Yaskawa INFORM job: X2_8B-21B(90,180)_HARDOX.JBI

/JOB
//NAME X2_8B-21B(90,180)_HARDOX
///FOLDERNAME X2
//POS
///NPOS 1745,1745,1745,47,0,0
///TOOL 0
///POSTYPE PULSE
///PULSE
C00000=-1415,-134459,-133802,-1969,12985,79332
C00001=-87080,-112473,-103627,-41798,51237,70410
C00002=-91681,-107347,-99471,-39221,49165,68848
C00003=-93439,-105106,-97054,-38371,48113,68361
C00004=-93441,-104864,-95967,-38672,47682,68565
C00005=-93504,-104969,-96260,-38564,47753,68495
C00006=-95585,-102642,-95415,-36914,47385,67494
C00007=-93504,-104969,-96260,-38564,47753,68495
C00008=-87147,-112175,-102116,-42180,50619,70689
C00009=-87145,-119394,-106475,-25944,48524,38750
C00010=-91166,-110510,-101811,-22693,48895,36705
C00011=-92650,-107060,-99920,-21494,49065,35962
C00012=-94767,-104655,-99060,-19829,49198,34943
C00013=-94484,-105085,-99259,-20052,49173,35080
C00014=-93721,-102513,-96995,-20598,49294,35408
C00015=-94484,-105085,-99259,-20052,49173,35080
C00016=-89209,-117497,-105909,-24366,48468,37757
C00017=-93166,-113214,-115710,-1969,57926,79332
C00018=-93710,-106990,-108704,-1652,56802,79139
C00019=-93766,-106412,-107148,-1629,56140,79127
C00020=-93768,-106433,-106329,-1638,55626,79135
C00021=-93918,-105383,-106173,-1535,56065,79069
C00022=-94164,-101296,-104676,-1361,57240,78956
C00023=-93895,-105502,-106499,-1547,56205,79076
C00024=-93151,-113316,-114305,-1998,57010,79354
C00025=-81072,-99391,-111155,-4750,63110,78553
C00026=-81984,-95120,-104767,-4287,61328,78293
C00027=-82103,-94682,-103397,-4241,60705,78273
C00028=-82106,-94924,-102383,-4271,59960,78300
C00029=-82089,-94934,-102578,-4276,60076,78302
C00030=-82803,-90374,-100753,-3806,61258,77993
C00031=-82089,-94934,-102578,-4276,60076,78302
C00032=-81057,-100006,-109908,-4804,62030,78604
C00033=-94004,-119945,-107122,49530,42714,48164
C00034=-93972,-116281,-97047,53343,39935,45878
C00035=-92833,-103149,-88492,51302,40218,47068
C00036=-93174,-100930,-87132,51219,40604,47120
C00037=-93174,-100493,-85792,51770,40220,46795
C00038=-93174,-101015,-87399,51095,40684,47186
C00039=-92955,-97894,-86230,50180,41136,47726
C00040=-93303,-100448,-87190,51023,40860,47230
C00041=-98055,-98607,-86499,53149,43882,46024
C00042=-96642,-96320,-85623,51883,43475,46780
C00043=-95342,-96864,-85830,51299,42647,47109
C00044=-97130,-98187,-86063,52744,43317,46271
C00045=-114545,-105110,-100746,39625,57097,48369
C00046=-113947,-102413,-97570,39574,56382,48359
C00047=-113947,-102278,-96691,39772,56015,48196
C00048=-113346,-99976,-96570,39024,56612,48763
C00049=-112899,-98120,-95866,38597,56823,49078
C00050=-114020,-99555,-96940,39169,57262,48705
C00051=-56302,-84822,-83054,-58022,66572,84014
C00052=-58361,-85953,-83540,-57558,65172,83717
C00053=-56302,-84822,-83054,-58022,66572,84014
C00054=-50122,-85714,-86741,-59061,71306,84454
C00055=-54195,-101901,-111197,-24063,62262,77343
C00056=-67243,-111926,-101536,21450,29925,69540
C00057=-66442,-101704,-94400,19916,30532,70304
C00058=-66308,-99858,-92576,19846,30336,70336
C00059=-66311,-99589,-91307,20230,29731,70137
C00060=-66308,-99960,-93112,19687,30597,70418
C00061=-70591,-100617,-92786,25268,31264,67678
C00062=-70591,-100325,-91437,25755,30647,67424
C00063=-68222,-99738,-91214,22742,30105,68906
C00064=-70591,-100606,-92729,25289,31242,67667
C00065=-66097,-110297,-96199,21577,27345,69446
C00066=-65719,-107666,-92844,21562,26575,69447
C00067=-65848,-106528,-92445,21497,26927,69482
C00068=-65365,-110699,-93884,21743,25627,69354
C00069=-67243,-111926,-101536,21450,29925,69540
C00070=-68963,-41843,-96211,-398,96948,-48811
C00071=-76932,-51697,-92360,2602,89609,-51106
C00072=-71886,-45093,-85416,705,88639,-49643
C00073=-71886,-45937,-84760,705,87803,-49648
C00074=-71886,-44632,-85753,705,89084,-49641
C00075=-68776,-90352,-95136,-4313,51281,-47645
C00076=-68803,-86754,-93636,-4241,52203,-47695
C00077=-68762,-92243,-95906,-4353,50785,-47617
C00078=-77446,-64871,-91176,8832,74282,-49527
C00079=-75907,-64612,-91046,8095,74185,-49034
C00080=-78150,-64967,-91224,9168,74335,-49752
C00081=-78150,-57569,-97635,8943,81990,-49191
C00082=-68963,-41843,-96211,-398,96948,-48811
C00083=-67385,-42511,-92598,-992,94393,-48367
C00084=-66773,-44328,-90253,-1220,92024,-48175
C00085=-66900,-44765,-89647,-1171,91425,-48205
C00086=-66773,-43962,-90441,-1221,92327,-48178
C00087=-69817,-49291,-93527,-72,91467,-49038
C00088=-102407,-61387,-79216,48101,75803,-74984
C00089=-99741,-62884,-79905,47237,74215,-74494
C00090=-102407,-61387,-79216,48101,75803,-74984
C00091=-71396,-101707,-96198,105,39560,-49678
C00092=-71544,-99303,-95354,247,40276,-49753
C00093=-71126,-105930,-97636,-165,38275,-49535
C00094=-74447,-120283,-111838,3099,39699,-51260
C00095=-57750,-84762,-113304,-22338,79933,-80646
C00096=-38298,-117376,-123136,-35520,84192,-83183
C00097=-31003,-114098,-105660,-45955,85390,-81321
C00098=-32496,-116782,-107403,-45795,84408,-81579
C00099=-34116,-118987,-108120,-45640,83088,-81742
C00100=-33779,-118873,-108083,-45678,83285,-81673
C00101=-33779,-118389,-106291,-45736,82677,-81394
C00102=-33116,-116007,-107005,-45711,84199,-81779
C00103=-43122,-77390,-91933,-43525,86904,-87571
C00104=-44353,-78017,-92219,-43231,86215,-87819
C00105=-45440,-79271,-92786,-42975,85486,-87990
C00106=-45102,-79332,-92813,-43057,85636,-87902
C00107=-45102,-79709,-91490,-43095,84888,-87585
C00108=-41853,-68825,-87871,-43817,88900,-87868
C00109=-48095,-31712,-66541,-47290,99218,-86920
C00110=-48762,-33638,-67810,-47108,98755,-86994
C00111=-49503,-35735,-69173,-46902,98237,-87073
C00112=-49389,-35416,-68966,-46933,98317,-87062
C00113=-49389,-36060,-68028,-46814,97684,-86756
C00114=-48487,-32850,-67294,-47182,98948,-86964
C00115=-45126,-25671,-76382,-49967,106798,-89554
C00116=-48508,-32956,-85951,-38791,109748,-85822
C00117=-73491,-115415,-129730,-12591,84406,-82629
C00118=-68604,-111632,-124361,34026,103601,-55041
C00119=-52690,-105642,-114364,31889,95098,-51390
C00120=-51347,-103959,-112740,31690,94497,-51045
C00121=-51347,-104280,-111882,31650,93903,-51212
C00122=-50963,-109237,-114816,31559,93129,-51281
C00123=-54701,-101748,-112541,32228,96580,-51739
C00124=-54580,-102143,-110625,32107,95358,-52042
C00125=-52710,-105778,-111943,31798,93771,-51772
C00126=-54580,-102143,-110625,32107,95358,-52042
C00127=-53574,-106836,-112314,31893,93817,-52092
C00128=-52008,-102475,-110737,31756,94333,-51344
C00129=-53574,-106836,-112314,31893,93817,-52092
C00130=-61074,-96775,-114868,33501,102293,-52496
C00131=-149084,-102156,-129577,22032,95315,-42360
C00132=-128569,-114069,-129208,14930,94899,-36248
C00133=-124702,-111484,-125119,14131,93099,-35189
C00134=-123206,-111006,-122572,13804,91571,-34868
C00135=-123205,-111346,-122108,13798,91123,-34918
C00136=-123169,-110975,-122344,13795,91444,-34870
C00137=-122647,-104244,-120003,13724,93323,-34489
C00138=-123169,-110975,-122344,13795,91444,-34870
C00139=-116503,-109521,-121739,12400,90787,-32743
C00140=-113941,-110266,-121994,11839,90202,-31960
C00141=-116503,-109521,-121739,12400,90787,-32743
C00142=-121595,-114825,-128025,13496,92670,-34216
C00143=-123984,-121300,-124584,22039,85383,-28695
C00144=-118596,-113071,-118409,20758,84424,-26972
C00145=-117828,-112575,-117002,20585,83663,-26833
C00146=-117596,-112721,-116348,20543,83158,-26838
C00147=-117643,-112201,-116474,20543,83493,-26797
C00148=-117846,-106122,-114344,20549,85245,-26570
C00149=-117643,-112201,-116474,20543,83493,-26797
C00150=-125192,-113488,-115877,22341,84450,-29296
C00151=-124919,-116220,-115928,22323,83104,-29449
C00152=-122352,-116155,-116251,21738,82647,-28614
C00153=-124919,-116220,-115928,22323,83104,-29449
C00154=-123984,-121300,-124584,22039,85383,-28695
C00155=-86442,-134681,-133724,-19248,79211,-32552
C00156=-86002,-121949,-124889,-19319,80358,-32581
C00157=-85994,-121959,-123892,-19351,79775,-32484
C00158=-85995,-122137,-123177,-19379,79272,-32404
C00159=-85938,-122450,-123568,-19392,79360,-32398
C00160=-86651,-115539,-121342,-19081,81262,-32951
C00161=-85938,-122450,-123568,-19392,79360,-32398
C00162=-130270,-119263,-121891,15868,79169,-48216
C00163=-132135,-133974,-122544,16883,72658,-49767
C00164=-129371,-136174,-123179,16117,71390,-48932
C00165=-132135,-133974,-122544,16883,72658,-49767
C00166=-120611,-122953,-119681,21560,80854,-22535
C00167=-120610,-122943,-118608,21593,80243,-22645
C00168=-120610,-122853,-116921,21650,79318,-22813
C00169=-120610,-122881,-117271,21638,79506,-22779
C00170=-120610,-122878,-117279,21638,79511,-22778
C00171=-120610,-122881,-117271,21638,79506,-22779
C00172=-120610,-122873,-117198,21640,79468,-22785
C00173=-120610,-122853,-117190,21640,79473,-22785
C00174=-120610,-122873,-117198,21640,79468,-22785
C00175=-120611,-122910,-120952,21522,81605,-22399
C00176=-120612,-120891,-127143,3106,87300,-4415
C00177=-120611,-122177,-124352,3111,84925,-4474
C00178=-120611,-122645,-122467,3116,83527,-4507
C00179=-120611,-122779,-121606,3119,82929,-4523
C00180=-120611,-122697,-122159,3117,83311,-4513
C00181=-120611,-122692,-122166,3117,83318,-4513
C00182=-120611,-122697,-122159,3117,83311,-4513
C00183=-120611,-121412,-126223,3107,86468,-4436
C00184=-96873,-136971,-131305,19961,95014,-27830
C00185=-53188,-122774,-119059,34227,101931,-42117
C00186=-53187,-122644,-116623,34032,100735,-42492
C00187=-53184,-122447,-115007,33919,99986,-42724
C00188=-53180,-122268,-113886,33849,99484,-42877
C00189=-53186,-122531,-115629,33961,100272,-42636
C00190=-53233,-122033,-113114,32057,113501,-44659
C00191=-53229,-122037,-113108,32057,113495,-44659
C00192=-53233,-122033,-113114,32057,113501,-44659
C00193=-53127,-122157,-112856,34567,84618,-41563
C00194=-53132,-122146,-112848,34568,84621,-41564
C00195=-53127,-122157,-112856,34567,84618,-41563
C00196=-53124,-122720,-116247,34514,86111,-41098
C00197=-68676,-133744,-131015,10578,108811,-68614
C00198=-80160,-118182,-130261,-41,125141,-81817
C00199=-80187,-122370,-123619,-70,118933,-81856
C00200=-80183,-122639,-122398,-68,118043,-81854
C00201=-80181,-122756,-121636,-67,117515,-81853
C00202=-80184,-122603,-122588,-68,118179,-81854
C00203=-80182,-122615,-122584,-67,118170,-81853
C00204=-80184,-122603,-122588,-68,118179,-81854
C00205=-80200,-121154,-126606,-75,121396,-81862
C00206=-109164,-117358,-132635,-7350,119146,-48306
C00207=-144183,-119511,-130571,-15498,107286,-7245
C00208=-197934,-122815,-127402,-28006,89082,55776
C00209=-202772,-123889,-124791,-27048,85608,54814
C00210=-204705,-124106,-122314,-26692,83530,54575
C00211=-204705,-124189,-120905,-26732,82711,54762
C00212=-205113,-122699,-120601,-26621,83104,54520
C00213=-208506,-122040,-120392,-25870,82241,53457
C00214=-204510,-125657,-121990,-26775,82699,54838
C00215=-204510,-125393,-124777,-26704,84359,54459
C00216=-217123,-144581,-130617,-26990,80795,43719
C00217=-208514,-157553,-136215,-22784,79668,13108
C00218=-208514,-151468,-127497,-22936,77598,13510
C00219=-209226,-147410,-126429,-22728,78719,13024
C00220=-208514,-151468,-127497,-22936,77598,13510
C00221=-208514,-156517,-134755,-22805,79329,13174
C00222=-187736,-116553,-120968,-36188,98329,31010
C00223=-144869,-104708,-130913,697,92502,-12445
C00224=-97478,-100538,-119508,25976,122096,-72949
C00225=-94415,-115583,-120723,24602,114867,-73486
C00226=-94145,-116737,-119872,24403,113768,-73630
C00227=-94090,-116915,-118863,24267,113100,-73760
C00228=-94227,-118887,-121662,24392,113788,-73658
C00229=-94618,-126072,-123928,23885,111795,-74261
C00230=-93811,-121058,-122280,24303,112998,-73673
C00231=-123165,-134656,-120887,30393,109989,-65140
C00232=-122877,-135920,-118822,30065,108215,-65520
C00233=-120918,-135771,-118381,30417,107339,-64954
C00234=-122877,-135920,-118822,30065,108215,-65520
C00235=-123434,-129548,-123417,31323,113703,-64157
C00236=-126606,-101457,-128935,16844,101795,-36174
C00237=-152779,-135138,-131563,2515,76140,-19155
C00238=-150820,-122490,-124749,1875,78392,-18455
C00239=-150097,-118368,-121531,1645,78513,-18212
C00240=-150095,-118599,-120646,1648,77850,-18220
C00241=-147666,-112236,-119185,871,80184,-17389
C00242=-146670,-110099,-118456,556,80825,-17059
C00243=-148658,-114325,-119887,1186,79554,-17722
C00244=-87079,-91764,-103818,-42328,107533,9448
C00245=-87027,-91004,-101788,-42122,106912,9740
C00246=-89264,-90509,-101588,-42089,105978,9119
C00247=-87027,-91004,-101788,-42122,106912,9740
C00248=-87391,-90282,-107909,-43186,109836,8282
C00249=-92115,-87061,-118989,-19004,94950,-3823
C00250=-78975,-130870,-123203,19746,71053,-12291
C00251=-74317,-97013,-111518,17407,83606,-9286
C00252=-74211,-95430,-110119,17377,83539,-9259
C00253=-74211,-95892,-109317,17397,82840,-9358
C00254=-75305,-113551,-114600,17838,69768,-10493
C00255=-78326,-111051,-111958,19079,70114,-11550
C00256=-78379,-106110,-110225,18937,71523,-11339
C00257=-78263,-116865,-113913,19272,68408,-11810
C00258=-85880,-113569,-112821,22054,71256,-14152
C00259=-85920,-114580,-110580,22309,69503,-14507
C00260=-82054,-114988,-110714,20879,68380,-13249
C00261=-85920,-114580,-110580,22309,69503,-14507
C00262=-78975,-130870,-123203,19746,67177,-12291
C00263=-159950,-115131,-126913,-23322,109234,64770
C00264=-163413,-124246,-126581,-22686,103792,64589
C00265=-164859,-127477,-125491,-22457,101245,64551
C00266=-164857,-127553,-124648,-22406,100728,64651
C00267=-164862,-127370,-126252,-22506,101730,64457
C00268=-158275,-145382,-129341,-21795,96649,67831
C00269=-159759,-153222,-131425,-21726,93697,67826
C00270=-158275,-145382,-129341,-21795,96649,67831
C00271=-157577,-144643,-126617,-21696,95625,68274
C00272=-160219,-140867,-125578,-21868,96138,67212
C00273=-157577,-144643,-126617,-21696,95625,68274
C00274=-152631,-134238,-128202,-21932,102817,68768
C00275=-146941,-123801,-133763,-3444,102850,52685
C00276=-136178,-116173,-124987,31736,84906,22811
C00277=-134413,-106132,-117362,31242,84680,23412
C00278=-134231,-105594,-115694,31219,83968,23286
C00279=-134230,-105863,-115134,31239,83552,23172
C00280=-134007,-104199,-114803,31151,84035,23389
C00281=-133473,-100630,-113499,30965,84737,23780
C00282=-134315,-106237,-115533,31260,83629,23161
C00283=-136272,-117460,-124003,31807,83855,22481
C00284=-136226,-116324,-125056,31750,84893,22789
C00285=-134474,-106353,-117504,31259,84679,23389
C00286=-134275,-105758,-115681,31235,83904,23252
C00287=-134274,-105987,-115198,31252,83547,23154
C00288=-134027,-104733,-115029,31162,83924,23350
C00289=-133465,-100971,-113658,30966,84667,23763
C00290=-134308,-106598,-115693,31262,83551,23142
C00291=-136269,-117902,-124178,31812,83752,22453
C00292=-139753,-124875,-130430,383,75663,-26245
C00293=-143223,-157944,-133481,-5653,58679,-38405
C00294=-140983,-144085,-126452,-6488,61628,-37698
C00295=-140148,-138933,-122655,-6835,62006,-37402
C00296=-140147,-138616,-121921,-6853,61719,-37384
C00297=-140691,-136506,-121897,-6553,62737,-37651
C00298=-138669,-131542,-120459,-7325,64564,-37004
C00299=-140691,-136506,-121897,-6553,62737,-37651
C00300=-145148,-139028,-124584,-4588,62787,-39337
C00301=-159973,-92454,-110285,14523,90938,-48717
C00302=-158765,-97223,-112137,14224,89465,-48492
C00303=-159973,-92454,-110285,14523,90938,-48717
C00304=-164681,-91509,-114703,15696,94847,-49769
C00305=-142525,-105883,-132766,-7713,103357,-60336
C00306=-90751,-115691,-121566,-36045,104861,-61043
C00307=-92920,-122587,-117773,-35137,99152,-60047
C00308=-93124,-123070,-117553,-35091,98753,-60003
C00309=-93124,-123008,-116878,-35050,98435,-59900
C00310=-93160,-123063,-117190,-35068,98555,-59953
C00311=-95752,-125144,-117838,-34977,96947,-60505
C00312=-93160,-123063,-117190,-35068,98555,-59953
C00313=-92038,-109836,-114685,-38536,89453,-57060
C00314=-86810,-100893,-104585,-47463,92019,-56975
C00315=-88449,-102594,-103600,-47188,90148,-56855
C00316=-88449,-102618,-102426,-47172,89639,-56610
C00317=-88449,-102603,-103366,-47184,90046,-56806
C00318=-85133,-99388,-102162,-47637,92393,-56350
C00319=-85168,-99488,-101153,-47595,91912,-56132
C00320=-86978,-101259,-101820,-47360,90627,-56378
C00321=-84037,-98201,-102123,-47804,93363,-56297
C00322=-108771,-112096,-123986,-16313,85813,-59347
C00323=-109769,-112695,-132242,-3132,99947,-61138
C00324=-127404,-127157,-120795,27540,73197,-60883
C00325=-120526,-123085,-115007,25540,69700,-59025
C00326=-119461,-122312,-114032,25210,69192,-58723
C00327=-119461,-122116,-113003,25293,68708,-58832
C00328=-119461,-122312,-114032,25210,69192,-58723
C00329=-94655,-112249,-115827,-1041,75214,-51009
C00330=-93364,-111129,-115444,-1499,75574,-50577
C00331=-121213,-123445,-114215,25873,69302,-59387
C00332=-127714,-127278,-119628,27738,72603,-61150
C00333=-140848,-129628,-128054,17424,84805,-27418
C00334=-127903,-106251,-120637,17388,91568,-15860
C00335=-124887,-98361,-114445,16717,91208,-14907
C00336=-124614,-94849,-112077,16660,91489,-14780
C00337=-117832,-103976,-115449,15062,87719,-13014
C00338=-118209,-109888,-118953,15141,86934,-13233
C00339=-120968,-118649,-124805,15800,86569,-14208
C00340=-112726,-101228,-128594,1890,90279,15897
C00341=-102865,-105549,-130121,-1361,88970,18873
C00342=-85416,-143080,-122146,-23399,58401,32529
C00343=-89847,-131888,-116792,-20882,59491,30436
C00344=-92125,-126361,-114096,-19602,60042,29398
C00345=-92108,-126361,-114086,-19611,60041,29405
C00346=-94963,-119193,-112807,-13876,65309,25883
C00347=-99230,-109273,-111594,-7832,72910,21884
C00348=-97558,-114678,-114533,-8498,72116,22521
C00349=-94805,-124749,-120489,-9597,70928,23580
C00350=-89899,-115674,-129227,-15589,81503,27304
C00351=-94000,-113154,-130859,1035,116659,-75004
C00352=-93721,-118000,-129934,5060,122177,-74127
C00353=-93715,-120352,-127357,4900,119392,-74256
C00354=-95346,-120435,-125547,4467,118331,-74923
C00355=-87734,-123112,-126247,6115,116903,-72103
C00356=-93725,-120284,-127319,4898,119404,-74259
C00357=-93731,-117931,-129895,5059,122189,-74130
C00358=-92605,-107385,-114202,-42080,118626,-78084
C00359=-94957,-117308,-114744,-40643,113912,-77125
C00360=-96859,-119647,-113709,-40343,111617,-77062
C00361=-96820,-119688,-113698,-40330,111613,-77042
C00362=-92369,-120637,-111842,-39132,112371,-75247
C00363=-87506,-133441,-114197,-38673,106213,-75021
C00364=-90618,-118755,-112828,-39302,114392,-75239
C00365=-88476,-109244,-112462,-40625,118981,-76164
C00366=-73726,-95231,-122050,-23824,117115,-78775
C00367=-68964,-113071,-130294,19412,109419,-80322
C00368=-55630,-112625,-122011,35520,97927,-81697
C00369=-52390,-118820,-120628,34805,93310,-81881
C00370=-47869,-106069,-116317,31727,98681,-78960
C00371=-58944,-112669,-113031,37596,97582,-82877
C00372=-56690,-122472,-119439,35129,92879,-83747
C00373=-59872,-116629,-120975,35716,97415,-83571
C00374=-61517,-148095,-119735,48293,75564,-80066
C00375=-55473,-148057,-116974,48060,71191,-79214
C00376=-53771,-146175,-114985,47935,70110,-78894
C00377=-54494,-144748,-112549,48210,69974,-79344
C00378=-55476,-147094,-115701,48129,70996,-79318
C00379=-61520,-147186,-118480,48348,75358,-80173
C00380=-69196,-132761,-125763,48066,87564,-77891
C00381=-67178,-112107,-133350,-9560,121946,-71499
C00382=-53652,-115588,-130730,-10921,119132,-80041
C00383=-53631,-118653,-128170,-10572,116038,-79726
C00384=-49406,-129162,-130962,-9295,109096,-77614
C00385=-56866,-119557,-126808,-10903,114346,-80761
C00386=-54665,-117852,-125979,-10629,114989,-80007
C00387=-57520,-119011,-127190,-3009,114777,-80027
C00388=-59278,-121853,-127991,842,113579,-80159
C00389=-55695,-120300,-124998,1328,112531,-78914
C00390=-53493,-120154,-126714,1639,113579,-78070
C00391=-53512,-117734,-129516,1682,116546,-78033
C00392=-64263,-112177,-127274,18013,116425,-52133
C00393=-53349,-113292,-116223,34708,105130,-41711
C00394=-53347,-113647,-113946,34435,103813,-42137
C00395=-52680,-112871,-112467,34368,103124,-42082
C00396=-58031,-122280,-112065,36284,98076,-45699
C00397=-53343,-113729,-112902,34324,103242,-42318
C00398=-53345,-113489,-115217,34581,104530,-41905
C00399=-83368,-135406,-127982,43757,111124,24122
C00400=-107112,-148704,-121184,48737,110155,73723
C00401=-107085,-142005,-111593,48000,108472,72828
C00402=-107084,-140010,-108705,47787,107957,72557
C00403=-87331,-137626,-115833,38185,104318,80918
C00404=-107143,-152743,-127540,-1092,113262,57657
C00405=-96955,-158208,-128899,-2670,111185,56030
C00406=-107130,-144670,-115956,-40497,90070,47196
C00407=-107133,-145289,-116877,-40503,90261,47122
C00408=-107139,-146938,-119316,-40521,90762,46927
C00409=-81304,-146505,-131302,-46256,99624,33732
C00410=-42290,-135810,-134986,-6789,56953,-43412
C00411=-53482,-111499,-99357,-5283,31563,-44884
C00412=-53488,-110753,-96932,-5448,30458,-44798
C00413=-53106,-110845,-96482,-5998,30161,-44520
C00414=-53143,-110117,-93832,-6189,28906,-44421
C00415=-53188,-109818,-93168,-6175,28651,-44427
C00416=-53095,-108922,-90553,-6542,27518,-44240
C00417=-53472,-108968,-91791,-5862,28222,-44586
C00418=-53466,-109889,-94290,-5675,29282,-44681
C00419=-93748,-113667,-111432,27227,62688,-41579
C00420=-93751,-113561,-109328,27520,61581,-41869
C00421=-94535,-110348,-107800,27711,62471,-41963
C00422=-94560,-109570,-102150,28499,59749,-42715
C00423=-93743,-112935,-104615,28181,59286,-42489
C00424=-93741,-113330,-106821,27872,60309,-42206
C00425=-53707,-103235,-126817,-3349,90409,-72793
C00426=-53694,-107630,-124107,-3352,86490,-72685
C00427=-53689,-108955,-122884,-3357,85060,-72645
C00428=-53697,-108940,-122873,-3354,85062,-72648
C00429=-53721,-108898,-122839,-3346,85062,-72656
C00430=-53729,-108884,-122827,-3345,85059,-72658
C00431=-53735,-107561,-124050,-3339,86489,-72698
C00432=-53748,-103173,-126762,-3336,90406,-72805
C00433=-44251,-68518,-112793,-6305,100072,-70363
C00434=-80270,30794,-42629,-11133,115571,-76543
C00435=-69737,67118,16632,-42575,112328,-80617
C00436=-69636,63823,22197,-49512,110599,-81416
C00437=-67564,55530,12856,-50142,112647,-81508
C00438=-66424,44944,1253,-49852,108764,-84350
C00439=-65618,29495,-14632,-48008,102670,-88237
C00440=-64581,15750,-27557,-48396,103780,-88326
C00441=-64160,11595,-31362,-48525,104124,-88308
C00442=-61878,-10748,-50140,-48981,105285,-87846
C00443=-62672,195,-41330,-51307,112408,-84907
C00444=-58944,10301,-35991,-52571,115494,-84879
C00445=-69716,-6230,-69222,-29298,97742,-75748
C00446=-102330,-22799,-82036,11222,88832,-73278
C00447=-48313,-118911,-129560,19207,92704,-27073
C00448=-53495,-110604,-121584,20154,93282,-28749
C00449=-53898,-112894,-120750,20179,91787,-29140
C00450=-54091,-109968,-119805,20238,92698,-29053
C00451=-54227,-109896,-119946,20266,92849,-29073
C00452=-54259,-112639,-122766,20278,93161,-29031
C00453=-53522,-108468,-123882,20258,95652,-28360
C00454=-66910,-101677,-117691,1645,82254,17515
C00455=-66905,-103395,-115374,1652,79946,17486
C00456=-66559,-103374,-114061,1536,79140,17588
C00457=-66525,-103141,-114029,1523,79241,17602
C00458=-67620,-103650,-114144,1902,79074,17240
C00459=-69811,-106122,-108316,12679,69437,17327
C00460=-66783,-105788,-110032,11324,70201,18483
C00461=-66785,-105108,-112553,11207,72068,18659
C00462=-34610,-119076,-126707,-31995,89279,47352
C00463=-26693,-119602,-105841,-51320,82883,62074
C00464=-26676,-118953,-103885,-51392,82336,62389
C00465=-26611,-118260,-103653,-51381,82509,62328
C00466=-26639,-116853,-99731,-51529,81413,62927
C00467=-26666,-118021,-101324,-51491,81640,62785
C00468=-26683,-118745,-103309,-51412,82173,62476
C00469=-26741,-121947,-116429,-51038,86269,60171
C00470=-80158,-111738,-121779,-46707,81282,-33331
C00471=-80124,-114295,-114082,-47454,77096,-31277
C00472=-80115,-114367,-110881,-47781,75720,-30584
C00473=-79927,-114969,-109893,-47987,75192,-30221
C00474=-79885,-115119,-109957,-48003,75187,-30197
C00475=-80052,-114603,-110983,-47806,75713,-30548
C00476=-80061,-114542,-114188,-47480,77086,-31241
C00477=-80063,-113108,-120040,-30435,104055,-77976
C00478=-80050,-114212,-116860,-30086,101864,-77373
C00479=-80380,-112077,-114717,-30053,101557,-77419
C00480=-79932,-114590,-112006,-35005,85347,-77215
C00481=-79912,-114566,-112044,-35008,85386,-77219
C00482=-80479,-112475,-109427,-36632,80098,-77307
C00483=-80029,-114714,-111597,-36713,80437,-77233
C00484=-82440,-93132,-104306,-35744,84828,-79668
C00485=-83378,-90315,-100640,-35536,83784,-79702
C00486=-86724,-76310,-94495,-34501,85296,-81493
C00487=-81341,-82881,-101909,-35963,88366,-80388
C00488=-80042,-114535,-115070,-36542,82240,-77847
C00489=-80040,-111621,-122742,-8414,85267,-41918
C00490=-80035,-113457,-119567,-8450,82400,-41723
C00491=-81798,-124774,-120168,-7328,73182,-41674
C00492=-80327,-109577,-118133,2572,87034,-53415
C00493=-79380,-112621,-119090,2349,86031,-53125
C00494=-78889,-114029,-118891,6085,83597,-58153
C00495=-80002,-113603,-119620,10752,83390,-63441
C00496=-80006,-103113,-128729,10775,94202,-62513
C00497=-39776,-103787,-110683,-21075,62663,59255
C00498=-39766,-104399,-107995,-21452,60825,59622
C00499=-41663,-99518,-106576,-17765,63773,58656
C00500=-39441,-104963,-106701,-21848,59898,59942
C00501=-39326,-105104,-106740,-21922,59881,59993
C00502=-39744,-104425,-108009,-21464,60826,59630
C00503=-39754,-103814,-110697,-21087,62664,59263
C00504=-47977,-106691,-119962,-23629,83327,62671
C00505=-66867,-99660,-121232,-22132,99220,62132
C00506=-66851,-102572,-118810,-21937,96446,62653
C00507=-74494,-137000,-128982,-14609,78071,53501
C00508=-72467,-138184,-128020,-15181,77278,54315
C00509=-67516,-140688,-126942,-16493,76361,56201
C00510=-43056,-127353,-114280,-36292,85121,62743
C00511=-66851,-103895,-117201,-21852,94891,62938
C00512=-66868,-101493,-119792,-22004,97521,62449
C00513=-74321,-107832,-126985,11736,80239,61811
C00514=-66584,-114412,-108983,34198,49386,64476
C00515=-66581,-113854,-105403,35147,47795,63826
C00516=-59001,-125725,-103773,32485,32454,61113
C00517=-65790,-113886,-101008,36132,45231,63145
C00518=-65568,-123466,-98279,45853,34675,56822
C00519=-65581,-123771,-97752,46366,34344,56544
C00520=-66567,-113311,-102857,35821,46729,63375
C00521=-66569,-114089,-106515,34851,48256,64025
C00522=-66614,-114312,-115902,32344,53032,65825
C00523=-26293,-124733,-123676,35115,86081,77095
C00524=-26278,-124914,-120130,35186,84196,76502
C00525=-26550,-125631,-118910,35285,83385,76132
C00526=-26140,-123752,-118256,35186,83681,76394
C00527=-26301,-124893,-120124,35190,84211,76498
C00528=-26317,-124710,-123669,35119,86096,77090
C00529=-26368,-124828,-121889,39154,95960,78120
C00530=-26350,-124746,-118556,38992,94373,77544
C00531=-26342,-124553,-116950,38932,93670,77290
C00532=-26340,-123995,-113991,38847,92461,76851
C00533=-26347,-124286,-115407,38884,93032,77056
C00534=-26365,-124761,-118865,39006,94524,77592
C00535=-26264,-124528,-116402,47920,86072,68134
C00536=-26249,-123768,-112787,47988,84810,67516
C00537=-26243,-123374,-111311,48022,84325,67278
C00538=-26226,-122772,-109280,48074,83674,66962
C00539=-26232,-123227,-110778,48035,84146,67194
C00540=-26247,-124165,-114452,47952,85370,67795
C00541=-82585,-123093,-118421,52491,64599,59558
C00542=-107155,-118824,-102398,58122,50036,52281
C00543=-107155,-117467,-98958,59145,49269,51564
C00544=-96813,-117817,-104188,42223,47347,50994
C00545=-105933,-121077,-109912,10415,42869,62990
C00546=-105953,-121074,-109843,10442,42831,62975
C00547=-107149,-121400,-109798,11502,42801,62375
C00548=-106717,-121349,-105974,7567,38238,71665
C00549=-107169,-120346,-107141,7797,39493,71540
C00550=-108433,-119625,-117514,7930,46308,71537
C00551=-107111,-122100,-111275,39348,45202,56077
C00552=-107109,-117760,-98763,43179,41028,53713
C00553=-106761,-117495,-97713,43363,40478,53604
C00554=-106458,-119074,-102370,12274,36991,61895
C00555=-94483,-118196,-102129,-13006,37418,75653
C00556=-107097,-114092,-90505,-56996,42891,80282
C00557=-107127,-114270,-91297,-56630,43098,80056
C00558=-101354,-119078,-102486,-55464,49091,79315
C00559=-93612,-109275,-133010,12113,75674,64968
C00560=-74458,-81913,-116300,25886,107898,47202
C00561=-74285,-84923,-113224,25351,104735,46539
C00562=-74085,-86300,-112083,25142,103399,46313
C00563=-71499,-76504,-108067,25490,106819,45523
C00564=-62961,-60085,-100217,24652,107848,48688
C00565=-60437,-59805,-99888,23461,105440,51393
C00566=-60588,-58283,-100875,23679,106756,51616
C00567=-60637,-54628,-103477,24231,109960,52288
C00568=-76657,-70403,-83915,51355,64349,40407
C00569=-74830,-68241,-74355,53953,55282,38932
C00570=-73110,-62379,-68708,53436,54020,39148
C00571=-73126,-62440,-68450,53549,53912,39057
C00572=-36930,-67607,-75173,-26029,44061,77403
C00573=-80523,-89058,-85253,18218,36719,55154
C00574=-82272,-90569,-85112,18702,34759,56728
C00575=-81508,-95500,-88175,18158,33969,56993
C00576=-81043,-103588,-94156,17854,33413,57140
C00577=-82846,-88179,-88219,41798,48730,43563
C00578=-81818,-81213,-82326,41198,48211,43888
C00579=-79663,-80074,-80946,37957,46333,45127
C00580=-64011,-84834,-85332,4259,39755,58703
C00581=-75846,-87347,-86370,15921,40584,52659
C00582=-47572,-67654,-78731,-37306,60592,66422
C00583=-46339,-68382,-80235,-37741,61555,66618
C00584=-42699,-70655,-83815,-39176,63943,67342
C00585=-43803,-67144,-92021,-36183,69839,64523
C00586=-86906,-70734,-117845,25978,101850,24881
C00587=-194376,-118372,-116958,36622,58194,-75254
C00588=-187943,-106127,-101715,33777,52366,-74665
C00589=-187951,-105693,-98645,34509,50978,-75202
C00590=-187954,-105458,-97394,34809,50440,-75417
C00591=-187960,-105469,-97402,34805,50444,-75420
C00592=-187927,-105629,-98482,19599,46235,-60273
C00593=-187923,-105820,-99644,19403,46817,-60144
C00594=-187914,-106157,-102495,18928,48312,-59826
C00595=-188021,-109107,-91072,54887,40419,-77132
C00596=-188025,-108188,-88773,55807,39869,-77674
C00597=-188027,-107805,-87846,56180,39654,-77892
C00598=-188036,-107761,-87717,56242,39627,-77928
C00599=-188035,-108145,-88644,55869,39841,-77710
C00600=-188030,-109068,-90945,54948,40390,-77168
C00601=-188015,-114130,-110744,41340,72657,-75143
C00602=-188018,-113864,-107763,41683,71368,-75679
C00603=-188019,-113684,-106544,41824,70871,-75888
C00604=-188009,-113674,-106577,41816,70886,-75877
C00605=-188008,-113852,-107795,41674,71383,-75668
C00606=-188005,-114114,-110775,41332,72673,-75132
C00607=-187933,-113872,-110928,18210,58720,-57176
C00608=-187882,-113256,-105308,-719,43762,-42538
C00609=-187896,-112711,-102669,-725,42418,-42533
C00610=-187852,-113170,-101841,-775,41671,-42505
C00611=-187778,-112374,-98354,-1639,37547,-42296
C00612=-187899,-111729,-99017,-1491,38283,-42378
C00613=-187886,-112431,-101600,-1465,39511,-42393
C00614=-192869,-127835,-120494,22551,66263,-53872
C00615=-188079,-122619,-114609,40714,83609,-61664
C00616=-188077,-122103,-112045,40794,82601,-62056
C00617=-188097,-121812,-110726,41966,87288,-59780
C00618=-188097,-121769,-110559,41966,87227,-59806
C00619=-188105,-121282,-108770,41980,86589,-60067
C00620=-188106,-121566,-109755,41972,86936,-59927
C00621=-188110,-122188,-112187,41960,87826,-59570
C00622=-188058,-121965,-125191,40549,88870,-59628
C00623=-104402,-90439,-123637,22599,88102,26907
C00624=-80407,-121901,-119741,18448,66455,46046
C00625=-80400,-121844,-116068,18757,64334,45697
C00626=-80358,-121826,-114599,18875,63477,45568
C00627=-79500,-120626,-114191,18436,63629,45929
C00628=-80475,-121542,-115946,18779,64427,45684
C00629=-80482,-121578,-119613,18469,66554,46034
C00630=-85156,-144709,-129107,-21632,59402,64028
C00631=-93856,-120445,-109825,-39450,57641,70752
C00632=-93847,-119691,-106928,-40019,56559,71233
C00633=-86628,-99816,-98593,-45940,69277,74290
C00634=-86043,-99167,-98859,-45014,69635,74495
C00635=-83318,-93529,-94650,-47165,68336,75996
C00636=-93680,-116508,-100417,-40719,46210,72415
C00637=-93820,-118277,-102341,-40471,46353,72255
C00638=-93828,-119232,-105178,-39715,47322,71755
C00639=-93822,-120125,-107980,-28359,52237,38282
C00640=-93816,-119582,-106091,-28689,51458,38525
C00641=-93813,-119346,-105328,-28822,51152,38622
C00642=-93805,-118409,-102529,-29499,49391,39302
C00643=-93820,-119862,-107056,-29266,59584,40856
C00644=-93823,-120114,-107958,-29147,59957,40747
C00645=-93830,-120670,-110185,-28854,60909,40473
C00646=-63807,-119595,-131717,-32346,77391,31957
C00647=-66677,-122882,-119460,-9954,65715,-31882
C00648=-66675,-122709,-116301,-10101,63887,-31721
C00649=-66675,-122586,-115330,-10147,63360,-31673
C00650=-66678,-122782,-121307,9429,81851,-37654
C00651=-66765,-122962,-121469,9451,81867,-37681
C00652=-66675,-122328,-113778,33290,107246,-42961
C00653=-66675,-122499,-114776,33395,107690,-42822
C00654=-66677,-122795,-117228,33681,108831,-42458
C00655=-66720,-122114,-124411,34847,112827,-41144
C00656=-15972,-110889,-128286,-10965,59905,-43045
C00657=-1415,-134459,-133802,-1969,12985,79332
C00658=-87080,-112473,-103627,-41798,51237,70410
C00659=-91681,-107347,-99471,-39221,49165,68848
C00660=-93439,-105106,-97054,-38371,48113,68361
C00661=-93441,-104864,-95967,-38672,47682,68565
C00662=-93504,-104969,-96260,-38564,47753,68495
C00663=-95585,-102642,-95415,-36914,47385,67494
C00664=-93504,-104969,-96260,-38564,47753,68495
C00665=-87147,-112175,-102116,-42180,50619,70689
C00666=-87145,-119394,-106475,-25944,48524,38750
C00667=-91166,-110510,-101811,-22693,48895,36705
C00668=-92650,-107060,-99920,-21494,49065,35962
C00669=-94767,-104655,-99060,-19829,49198,34943
C00670=-94484,-105085,-99259,-20052,49173,35080
C00671=-93721,-102513,-96995,-20598,49294,35408
C00672=-94484,-105085,-99259,-20052,49173,35080
C00673=-89209,-117497,-105909,-24366,48468,37757
C00674=-93166,-113214,-115710,-1969,57926,79332
C00675=-122366,-117496,-112293,16338,56235,67679
C00676=-123456,-103417,-106445,16337,59944,67813
C00677=-123456,-103539,-105172,16474,59132,67689
C00678=-123456,-103531,-105272,16463,59195,67698
C00679=-123128,-98284,-103303,16044,60561,68033
C00680=-123156,-99911,-105489,15984,61057,68095
C00681=-93710,-106990,-108704,-1652,56802,79139
C00682=-93766,-106412,-107148,-1629,56140,79127
C00683=-93768,-106433,-106329,-1638,55626,79135
C00684=-93918,-105383,-106173,-1535,56065,79069
C00685=-94164,-101296,-104676,-1361,57240,78956
C00686=-93895,-105502,-106499,-1547,56205,79076
C00687=-93151,-113316,-114305,-1998,57010,79354
C00688=-81072,-99391,-111155,-4750,63110,78553
C00689=-81984,-95120,-104767,-4287,61328,78293
C00690=-82103,-94682,-103397,-4241,60705,78273
C00691=-82106,-94924,-102383,-4271,59960,78300
C00692=-82089,-94934,-102578,-4276,60076,78302
C00693=-82803,-90374,-100753,-3806,61258,77993
C00694=-82089,-94934,-102578,-4276,60076,78302
C00695=-81057,-100006,-109908,-4804,62030,78604
C00696=-94004,-119945,-107122,49530,42714,48164
C00697=-93972,-116281,-97047,53343,39935,45878
C00698=-92833,-103149,-88492,51302,40218,47068
C00699=-93174,-100930,-87132,51219,40604,47120
C00700=-93174,-100493,-85792,51770,40220,46795
C00701=-93174,-101015,-87399,51095,40684,47186
C00702=-92955,-97894,-86230,50180,41136,47726
C00703=-93303,-100448,-87190,51023,40860,47230
C00704=-98055,-98607,-86499,53149,43882,46024
C00705=-96642,-96320,-85623,51883,43475,46780
C00706=-95342,-96864,-85830,51299,42647,47109
C00707=-97130,-98187,-86063,52744,43317,46271
C00708=-114545,-105110,-100746,39625,57097,48369
C00709=-113947,-102413,-97570,39574,56382,48359
C00710=-113947,-102278,-96691,39772,56015,48196
C00711=-113346,-99976,-96570,39024,56612,48763
C00712=-112899,-98120,-95866,38597,56823,49078
C00713=-114020,-99555,-96940,39169,57262,48705
C00714=-56302,-84822,-83054,-58022,66572,84014
C00715=-58361,-85953,-83540,-57558,65172,83717
C00716=-56302,-84822,-83054,-58022,66572,84014
C00717=-50122,-85714,-86741,-59061,71306,84454
C00718=-54195,-101901,-111197,-24063,62262,77343
C00719=-67243,-111926,-101536,21450,29925,69540
C00720=-66442,-101704,-94400,19916,30532,70304
C00721=-66308,-99858,-92576,19846,30336,70336
C00722=-66311,-99589,-91307,20230,29731,70137
C00723=-66308,-99960,-93112,19687,30597,70418
C00724=-70591,-100617,-92786,25268,31264,67678
C00725=-70591,-100325,-91437,25755,30647,67424
C00726=-68222,-99738,-91214,22742,30105,68906
C00727=-70591,-100606,-92729,25289,31242,67667
C00728=-66097,-110297,-96199,21577,27345,69446
C00729=-65719,-107666,-92844,21562,26575,69447
C00730=-65848,-106528,-92445,21497,26927,69482
C00731=-65365,-110699,-93884,21743,25627,69354
C00732=-67243,-111926,-101536,21450,29925,69540
C00733=-68963,-41843,-96211,-398,96948,-48811
C00734=-76932,-51697,-92360,2602,89609,-51106
C00735=-71886,-45093,-85416,705,88639,-49643
C00736=-71886,-45937,-84760,705,87803,-49648
C00737=-71886,-44632,-85753,705,89084,-49641
C00738=-68776,-90352,-95136,-4313,51281,-47645
C00739=-68803,-86754,-93636,-4241,52203,-47695
C00740=-68762,-92243,-95906,-4353,50785,-47617
C00741=-77446,-64871,-91176,8832,74282,-49527
C00742=-75907,-64612,-91046,8095,74185,-49034
C00743=-78150,-64967,-91224,9168,74335,-49752
C00744=-78150,-57569,-97635,8943,81990,-49191
C00745=-68963,-41843,-96211,-398,96948,-48811
C00746=-67385,-42511,-92598,-992,94393,-48367
C00747=-66773,-44328,-90253,-1220,92024,-48175
C00748=-66900,-44765,-89647,-1171,91425,-48205
C00749=-66773,-43962,-90441,-1221,92327,-48178
C00750=-69817,-49291,-93527,-72,91467,-49038
C00751=-102407,-61387,-79216,48101,75803,-74984
C00752=-99741,-62884,-79905,47237,74215,-74494
C00753=-102407,-61387,-79216,48101,75803,-74984
C00754=-71396,-101707,-96198,105,39560,-49678
C00755=-71544,-99303,-95354,247,40276,-49753
C00756=-71126,-105930,-97636,-165,38275,-49535
C00757=-74447,-120283,-111838,3099,39699,-51260
C00758=-57750,-84762,-113304,-22338,79933,-80646
C00759=-38298,-117376,-123136,-35520,84192,-83183
C00760=-31003,-114098,-105660,-45955,85390,-81321
C00761=-32496,-116782,-107403,-45795,84408,-81579
C00762=-34116,-118987,-108120,-45640,83088,-81742
C00763=-33779,-118873,-108083,-45678,83285,-81673
C00764=-33779,-118389,-106291,-45736,82677,-81394
C00765=-33116,-116007,-107005,-45711,84199,-81779
C00766=-43122,-77390,-91933,-43525,86904,-87571
C00767=-44353,-78017,-92219,-43231,86215,-87819
C00768=-45440,-79271,-92786,-42975,85486,-87990
C00769=-45102,-79332,-92813,-43057,85636,-87902
C00770=-45102,-79709,-91490,-43095,84888,-87585
C00771=-41853,-68825,-87871,-43817,88900,-87868
C00772=-48095,-31712,-66541,-47290,99218,-86920
C00773=-48762,-33638,-67810,-47108,98755,-86994
C00774=-49503,-35735,-69173,-46902,98237,-87073
C00775=-49389,-35416,-68966,-46933,98317,-87062
C00776=-49389,-36060,-68028,-46814,97684,-86756
C00777=-48487,-32850,-67294,-47182,98948,-86964
C00778=-45126,-25671,-76382,-49967,106798,-89554
C00779=-48508,-32956,-85951,-38791,109748,-85822
C00780=-73491,-115415,-129730,-12591,84406,-82629
C00781=-68604,-111632,-124361,34026,103601,-55041
C00782=-52690,-105642,-114364,31889,95098,-51390
C00783=-50963,-109289,-114635,31553,93010,-51314
C00784=-50968,-109442,-114037,31534,92627,-51422
C00785=-50963,-109237,-114816,31559,93129,-51281
C00786=-54701,-101748,-112541,32228,96580,-51739
C00787=-54580,-102143,-110625,32107,95358,-52042
C00788=-52710,-105778,-111943,31798,93771,-51772
C00789=-54580,-102143,-110625,32107,95358,-52042
C00790=-53574,-106836,-112314,31893,93817,-52092
C00791=-52008,-102475,-110737,31756,94333,-51344
C00792=-53574,-106836,-112314,31893,93817,-52092
C00793=-61074,-96775,-114868,33501,102293,-52496
C00794=-149084,-102156,-129577,22032,95315,-42360
C00795=-128569,-114069,-129208,14930,94899,-36248
C00796=-124702,-111484,-125119,14131,93099,-35189
C00797=-123206,-111006,-122572,13804,91571,-34868
C00798=-123205,-111346,-122108,13798,91123,-34918
C00799=-123169,-110975,-122344,13795,91444,-34870
C00800=-122647,-104244,-120003,13724,93323,-34489
C00801=-123169,-110975,-122344,13795,91444,-34870
C00802=-116503,-109521,-121739,12400,90787,-32743
C00803=-113941,-110266,-121994,11839,90202,-31960
C00804=-116503,-109521,-121739,12400,90787,-32743
C00805=-121595,-114825,-128025,13496,92670,-34216
C00806=-123984,-121300,-124584,22039,85383,-28695
C00807=-118596,-113071,-118409,20758,84424,-26972
C00808=-117828,-112575,-117002,20585,83663,-26833
C00809=-117596,-112721,-116348,20543,83158,-26838
C00810=-117643,-112201,-116474,20543,83493,-26797
C00811=-117846,-106122,-114344,20549,85245,-26570
C00812=-117643,-112201,-116474,20543,83493,-26797
C00813=-125192,-113488,-115877,22341,84450,-29296
C00814=-124919,-116220,-115928,22323,83104,-29449
C00815=-122352,-116155,-116251,21738,82647,-28614
C00816=-124919,-116220,-115928,22323,83104,-29449
C00817=-123984,-121300,-124584,22039,85383,-28695
C00818=-86442,-134681,-133724,-19248,79211,-32552
C00819=-86002,-121949,-124889,-19319,80358,-32581
C00820=-85994,-121959,-123892,-19351,79775,-32484
C00821=-85995,-122137,-123177,-19379,79272,-32404
C00822=-85938,-122450,-123568,-19392,79360,-32398
C00823=-86651,-115539,-121342,-19081,81262,-32951
C00824=-85938,-122450,-123568,-19392,79360,-32398
C00825=-130270,-119263,-121891,15868,79169,-48216
C00826=-132135,-133974,-122544,16883,72658,-49767
C00827=-129371,-136174,-123179,16117,71390,-48932
C00828=-132135,-133974,-122544,16883,72658,-49767
C00829=-120611,-122953,-119681,21560,80854,-22535
C00830=-120610,-122943,-118608,21593,80243,-22645
C00831=-120610,-122853,-116921,21650,79318,-22813
C00832=-120610,-122881,-117271,21638,79506,-22779
C00833=-120610,-122878,-117279,21638,79511,-22778
C00834=-120610,-122881,-117271,21638,79506,-22779
C00835=-120610,-122873,-117198,21640,79468,-22785
C00836=-120610,-122853,-117190,21640,79473,-22785
C00837=-120610,-122873,-117198,21640,79468,-22785
C00838=-120611,-122910,-120952,21522,81605,-22399
C00839=-86002,-120340,-127953,-19212,82925,-32989
C00840=-85994,-121959,-123892,-19351,79775,-32484
C00841=-85995,-122137,-123177,-19379,79272,-32404
C00842=-85938,-122450,-123568,-19392,79360,-32398
C00843=-86651,-115539,-121342,-19081,81262,-32951
C00844=-85938,-122450,-123568,-19392,79360,-32398
C00845=-130270,-119263,-121891,15868,79169,-48216
C00846=-132135,-133974,-122544,16883,72658,-49767
C00847=-129371,-136174,-123179,16117,71390,-48932
C00848=-132135,-133974,-122544,16883,72658,-49767
C00849=-120612,-120891,-127143,3106,87300,-4415
C00850=-120611,-122177,-124352,3111,84925,-4474
C00851=-120611,-122645,-122467,3116,83527,-4507
C00852=-120611,-122779,-121606,3119,82929,-4523
C00853=-120611,-122697,-122159,3117,83311,-4513
C00854=-120611,-122692,-122166,3117,83318,-4513
C00855=-120611,-122697,-122159,3117,83311,-4513
C00856=-120611,-121412,-126223,3107,86468,-4436
C00857=-120611,-118807,-129728,3107,89959,-4350
C00858=-120605,-132560,-136700,3104,87187,-4416
C00859=-53188,-122658,-121398,34453,103181,-41719
C00860=-53187,-122644,-116623,34032,100735,-42492
C00861=-53184,-122447,-115007,33919,99986,-42724
C00862=-53180,-122268,-113886,33849,99484,-42877
C00863=-53186,-122531,-115629,33961,100272,-42636
C00864=-53233,-122033,-113114,32057,113501,-44659
C00865=-53229,-122037,-113108,32057,113495,-44659
C00866=-53233,-122033,-113114,32057,113501,-44659
C00867=-53127,-122157,-112856,34567,84618,-41563
C00868=-53132,-122146,-112848,34568,84621,-41564
C00869=-53127,-122157,-112856,34567,84618,-41563
C00870=-53124,-122720,-116247,34514,86111,-41098
C00871=-61684,-126457,-131749,21672,103686,-55019
C00872=-68676,-133744,-131015,10578,108811,-68614
C00873=-80160,-118182,-130261,-41,125141,-81817
C00874=-80187,-122370,-123619,-70,118933,-81856
C00875=-80183,-122639,-122398,-68,118043,-81854
C00876=-80181,-122756,-121636,-67,117515,-81853
C00877=-80184,-122603,-122588,-68,118179,-81854
C00878=-80182,-122615,-122584,-67,118170,-81853
C00879=-80184,-122603,-122588,-68,118179,-81854
C00880=-80200,-121154,-126606,-75,121396,-81862
C00881=-109164,-117358,-132635,-7350,119146,-48306
C00882=-144183,-119511,-130571,-15498,107286,-7245
C00883=-197934,-122815,-127402,-28006,89082,55776
C00884=-202772,-123889,-124791,-27048,85608,54814
C00885=-204705,-124106,-122314,-26692,83530,54575
C00886=-204705,-124189,-120905,-26732,82711,54762
C00887=-205113,-122699,-120601,-26621,83104,54520
C00888=-208506,-122040,-120392,-25870,82241,53457
C00889=-204510,-125657,-121990,-26775,82699,54838
C00890=-204510,-125393,-124777,-26704,84359,54459
C00891=-217123,-144581,-130617,-26990,80795,43719
C00892=-208514,-157553,-136215,-22784,79668,13108
C00893=-208134,-153606,-128050,-23049,77001,13769
C00894=-209226,-147410,-126429,-22728,78719,13024
C00895=-208514,-151468,-127497,-22936,77598,13510
C00896=-208514,-156517,-134755,-22805,79329,13174
C00897=-197934,-122815,-127402,-28006,89082,55776
C00898=-202772,-123889,-124791,-27048,85608,54814
C00899=-204705,-124106,-122314,-26692,83530,54575
C00900=-204705,-124189,-120905,-26732,82711,54762
C00901=-205113,-122699,-120601,-26621,83104,54520
C00902=-208506,-122040,-120392,-25870,82241,53457
C00903=-204510,-125657,-121990,-26775,82699,54838
C00904=-204510,-125393,-124777,-26704,84359,54459
C00905=-217123,-144581,-130617,-26990,80795,43719
C00906=-216657,-144339,-132121,-20327,83655,24427
C00907=-208514,-151468,-127497,-22936,77598,13510
C00908=-209226,-147410,-126429,-22728,78719,13024
C00909=-208514,-151468,-127497,-22936,77598,13510
C00910=-208514,-156517,-134755,-22805,79329,13174
C00911=-187736,-116553,-120968,-36188,98329,31010
C00912=-144869,-104708,-130913,697,92502,-12445
C00913=-97478,-100538,-119508,25976,122096,-72949
C00914=-94415,-115583,-120723,24602,114867,-73486
C00915=-94145,-116737,-119872,24403,113768,-73630
C00916=-94090,-116915,-118863,24267,113100,-73760
C00917=-94227,-118887,-121662,24392,113788,-73658
C00918=-94618,-126072,-123928,23885,111795,-74261
C00919=-93811,-121058,-122280,24303,112998,-73673
C00920=-123165,-134656,-120887,30393,109989,-65140
C00921=-122877,-135920,-118822,30065,108215,-65520
C00922=-120918,-135771,-118381,30417,107339,-64954
C00923=-122877,-135920,-118822,30065,108215,-65520
C00924=-123434,-129548,-123417,31323,113703,-64157
C00925=-126606,-101457,-128935,16844,101795,-36174
C00926=-152779,-135138,-131563,2515,76140,-19155
C00927=-150820,-122490,-124749,1875,78392,-18455
C00928=-150097,-118368,-121531,1645,78513,-18212
C00929=-150095,-118599,-120646,1648,77850,-18220
C00930=-147666,-112236,-119185,871,80184,-17389
C00931=-146670,-110099,-118456,556,80825,-17059
C00932=-148658,-114325,-119887,1186,79554,-17722
C00933=-87079,-91764,-103818,-42328,107533,9448
C00934=-87027,-91004,-101788,-42122,106912,9740
C00935=-89264,-90509,-101588,-42089,105978,9119
C00936=-87027,-91004,-101788,-42122,106912,9740
C00937=-87391,-90282,-107909,-43186,109836,8282
C00938=-92115,-87061,-118989,-19004,94950,-3823
C00939=-78975,-130870,-123203,19746,71053,-12291
C00940=-74317,-97013,-111518,17407,83606,-9286
C00941=-74211,-95430,-110119,17377,83539,-9259
C00942=-74211,-95892,-109317,17397,82840,-9358
C00943=-75305,-113551,-114600,17838,69768,-10493
C00944=-78326,-111051,-111958,19079,70114,-11550
C00945=-78379,-106110,-110225,18937,71523,-11339
C00946=-78263,-116865,-113913,19272,68408,-11810
C00947=-85880,-113569,-112821,22054,71256,-14152
C00948=-85920,-114580,-110580,22309,69503,-14507
C00949=-82054,-114988,-110714,20879,68380,-13249
C00950=-85920,-114580,-110580,22309,69503,-14507
C00951=-78975,-130870,-123203,19746,67177,-12291
C00952=-159950,-115131,-126913,-23322,109234,64770
C00953=-163413,-124246,-126581,-22686,103792,64589
C00954=-164859,-127477,-125491,-22457,101245,64551
C00955=-164857,-127553,-124648,-22406,100728,64651
C00956=-164862,-127370,-126252,-22506,101730,64457
C00957=-158275,-145382,-129341,-21795,96649,67831
C00958=-159759,-153222,-131425,-21726,93697,67826
C00959=-158275,-145382,-129341,-21795,96649,67831
C00960=-157577,-144643,-126617,-21696,95625,68274
C00961=-160219,-140867,-125578,-21868,96138,67212
C00962=-157577,-144643,-126617,-21696,95625,68274
C00963=-152631,-134238,-128202,-21932,102817,68768
C00964=-146941,-123801,-133763,-3444,102850,52685
C00965=-136178,-116173,-124987,31736,84906,22811
C00966=-134413,-106132,-117362,31242,84680,23412
C00967=-134231,-105594,-115694,31219,83968,23286
C00968=-134230,-105863,-115134,31239,83552,23172
C00969=-134007,-104199,-114803,31151,84035,23389
C00970=-133473,-100630,-113499,30965,84737,23780
C00971=-134315,-106237,-115533,31260,83629,23161
C00972=-136272,-117460,-124003,31807,83855,22481
C00973=-136226,-116324,-125056,31750,84893,22789
C00974=-134474,-106353,-117504,31259,84679,23389
C00975=-134275,-105758,-115681,31235,83904,23252
C00976=-134274,-105987,-115198,31252,83547,23154
C00977=-134027,-104733,-115029,31162,83924,23350
C00978=-133465,-100971,-113658,30966,84667,23763
C00979=-134308,-106598,-115693,31262,83551,23142
C00980=-178993,-121773,-123174,38769,99022,10273
C00981=-175539,-115427,-119854,38657,98481,11541
C00982=-175539,-115857,-118311,38525,97555,11203
C00983=-175539,-115829,-118427,38535,97623,11227
C00984=-173168,-111114,-116839,38478,97741,12267
C00985=-174072,-113112,-119760,38657,98741,12252
C00986=-136269,-117902,-124178,31812,83752,22453
C00987=-139753,-124875,-130430,383,75663,-26245
C00988=-143223,-157944,-133481,-5653,58679,-38405
C00989=-140983,-144085,-126452,-6488,61628,-37698
C00990=-140148,-138933,-122655,-6835,62006,-37402
C00991=-140147,-138616,-121921,-6853,61719,-37384
C00992=-140691,-136506,-121897,-6553,62737,-37651
C00993=-138669,-131542,-120459,-7325,64564,-37004
C00994=-140691,-136506,-121897,-6553,62737,-37651
C00995=-145148,-139028,-124584,-4588,62787,-39337
C00996=-159973,-92454,-110285,14523,90938,-48717
C00997=-158765,-97223,-112137,14224,89465,-48492
C00998=-159973,-92454,-110285,14523,90938,-48717
C00999=-164681,-91509,-114703,15696,94847,-49769
C01000=-142525,-105883,-132766,-7713,103357,-60336
C01001=-90751,-115691,-121566,-36045,104861,-61043
C01002=-92920,-122587,-117773,-35137,99152,-60047
C01003=-93124,-123070,-117553,-35091,98753,-60003
C01004=-93124,-123008,-116878,-35050,98435,-59900
C01005=-93160,-123063,-117190,-35068,98555,-59953
C01006=-95752,-125144,-117838,-34977,96947,-60505
C01007=-93160,-123063,-117190,-35068,98555,-59953
C01008=-92038,-109836,-114685,-38536,89453,-57060
C01009=-86810,-100893,-104585,-47463,92019,-56975
C01010=-88449,-102594,-103600,-47188,90148,-56855
C01011=-88449,-102618,-102426,-47172,89639,-56610
C01012=-88449,-102603,-103366,-47184,90046,-56806
C01013=-85133,-99388,-102162,-47637,92393,-56350
C01014=-85168,-99488,-101153,-47595,91912,-56132
C01015=-86978,-101259,-101820,-47360,90627,-56378
C01016=-84037,-98201,-102123,-47804,93363,-56297
C01017=-108771,-112096,-123986,-16313,85813,-59347
C01018=-109769,-112695,-132242,-3132,99947,-61138
C01019=-127404,-127157,-120795,27540,73197,-60883
C01020=-120526,-123085,-115007,25540,69700,-59025
C01021=-119461,-122312,-114032,25210,69192,-58723
C01022=-119461,-122116,-113003,25293,68708,-58832
C01023=-119461,-122312,-114032,25210,69192,-58723
C01024=-94655,-112249,-115827,-1041,75214,-51009
C01025=-93364,-111129,-115444,-1499,75574,-50577
C01026=-121213,-123445,-114215,25873,69302,-59387
C01027=-127714,-127278,-119628,27738,72603,-61150
C01028=-140848,-129628,-128054,17424,84805,-27418
C01029=-127903,-106251,-120637,17388,91568,-15860
C01030=-124887,-98361,-114445,16717,91208,-14907
C01031=-124532,-94860,-112080,16625,91471,-14753
C01032=-117832,-103976,-115449,15062,87719,-13014
C01033=-118209,-109888,-118953,15141,86934,-13233
C01034=-120968,-118649,-124805,15800,86569,-14208
C01035=-112726,-101228,-128594,1890,90279,15897
C01036=-102865,-105549,-130121,-1361,88970,18873
C01037=-85416,-143080,-122146,-23399,58401,32529
C01038=-89847,-131888,-116792,-20882,59491,30436
C01039=-92125,-126361,-114096,-19602,60042,29398
C01040=-92108,-126361,-114086,-19611,60041,29405
C01041=-94963,-119193,-112807,-13876,65309,25883
C01042=-99230,-109273,-111594,-7832,72910,21884
C01043=-97558,-114678,-114533,-8498,72116,22521
C01044=-94805,-124749,-120489,-9597,70928,23580
C01045=-89899,-115674,-129227,-15589,81503,27304
C01046=-94000,-113154,-130859,1035,116659,-75004
C01047=-93721,-118000,-129934,5060,122177,-74127
C01048=-93715,-120352,-127357,4900,119392,-74256
C01049=-95346,-120435,-125547,4467,118331,-74923
C01050=-87734,-123112,-126247,6115,116903,-72103
C01051=-93725,-120284,-127319,4898,119404,-74259
C01052=-93731,-117931,-129895,5059,122189,-74130
C01053=-92605,-107385,-114202,-42080,118626,-78084
C01054=-94957,-117308,-114744,-40643,113912,-77125
C01055=-96859,-119647,-113709,-40343,111617,-77062
C01056=-96820,-119688,-113698,-40330,111613,-77042
C01057=-92369,-120637,-111842,-39132,112371,-75247
C01058=-87506,-133441,-114197,-38673,106213,-75021
C01059=-90618,-118755,-112828,-39302,114392,-75239
C01060=-88476,-109244,-112462,-40625,118981,-76164
C01061=-73726,-95231,-122050,-23824,117115,-78775
C01062=-68964,-113071,-130294,19412,109419,-80322
C01063=-55630,-112625,-122011,35520,97927,-81697
C01064=-52390,-118820,-120628,34805,93310,-81881
C01065=-53603,-103093,-112884,36459,100480,-79984
C01066=-59619,-117562,-114740,37336,94951,-84077
C01067=-56690,-122472,-119439,35129,92879,-83747
C01068=-59872,-116629,-120975,35716,97415,-83571
C01069=-61517,-148095,-119735,48293,75564,-80066
C01070=-55473,-148057,-116974,48060,71191,-79214
C01071=-53771,-146175,-114985,47935,70110,-78894
C01072=-54494,-144748,-112549,48210,69974,-79344
C01073=-55476,-147094,-115701,48129,70996,-79318
C01074=-61520,-147186,-118480,48348,75358,-80173
C01075=-87978,-108563,-128727,6750,125872,-71649
C01076=-93715,-120352,-127357,4900,119392,-74256
C01077=-94748,-123674,-126724,4558,117361,-74733
C01078=-87347,-125535,-127084,6155,116151,-72000
C01079=-93725,-120284,-127319,4898,119404,-74259
C01080=-93731,-117931,-129895,5059,122189,-74130
C01081=-92605,-107385,-114202,-42080,118626,-78084
C01082=-94957,-117308,-114744,-40643,113912,-77125
C01083=-96514,-122009,-114462,-40074,111194,-76723
C01084=-96015,-122145,-114253,-39942,111269,-76518
C01085=-92174,-122830,-112540,-38890,111906,-74970
C01086=-86945,-136787,-114983,-38317,105485,-74493
C01087=-90618,-118755,-112828,-39302,114392,-75239
C01088=-88476,-109244,-112462,-40625,118981,-76164
C01089=-73726,-95231,-122050,-23824,117115,-78775
C01090=-68964,-113071,-130294,19412,109419,-80322
C01091=-55630,-112625,-122011,35520,97927,-81697
C01092=-52390,-118820,-120628,34805,93310,-81881
C01093=-47304,-107066,-116669,31636,98225,-78870
C01094=-58547,-113359,-113266,37552,97245,-82829
C01095=-56690,-122472,-119439,35129,92879,-83747
C01096=-59872,-116629,-120975,35716,97415,-83571
C01097=-61517,-148095,-119735,48293,75564,-80066
C01098=-55473,-148057,-116974,48060,71191,-79214
C01099=-53043,-147267,-115261,47953,69457,-78858
C01100=-53748,-146178,-113424,48182,69442,-79233
C01101=-55476,-147094,-115701,48129,70996,-79318
C01102=-61520,-147186,-118480,48348,75358,-80173
C01103=-69196,-132761,-125763,48066,87564,-77891
C01104=-67178,-112107,-133350,-9560,121946,-71499
C01105=-53652,-115588,-130730,-10921,119132,-80041
C01106=-53631,-118653,-128170,-10572,116038,-79726
C01107=-49406,-129162,-130962,-9295,109096,-77614
C01108=-56866,-119557,-126808,-10903,114346,-80761
C01109=-54665,-117852,-125979,-10629,114989,-80007
C01110=-57520,-119011,-127190,-3009,114777,-80027
C01111=-59278,-121853,-127991,842,113579,-80159
C01112=-55695,-120300,-124998,1328,112531,-78914
C01113=-53493,-120154,-126714,1639,113579,-78070
C01114=-53512,-117734,-129516,1682,116546,-78033
C01115=-64263,-112177,-127274,18013,116425,-52133
C01116=-53349,-113292,-116223,34708,105130,-41711
C01117=-53347,-113647,-113946,34435,103813,-42137
C01118=-52680,-112871,-112467,34368,103124,-42082
C01119=-58031,-122280,-112065,36284,98076,-45699
C01120=-53343,-113729,-112902,34324,103242,-42318
C01121=-53345,-113489,-115217,34581,104530,-41905
C01122=-83368,-135406,-127982,43757,111124,24122
C01123=-107112,-148704,-121184,48737,110155,73723
C01124=-107085,-142005,-111593,48000,108472,72828
C01125=-107084,-140010,-108705,47787,107957,72557
C01126=-87331,-137626,-115833,38185,104318,80918
C01127=-107143,-152743,-127540,-1092,113262,57657
C01128=-106498,-152435,-127519,-1673,113318,57021
C01129=-107059,-148801,-134211,-1989,119286,56706
C01130=-109333,-147161,-118098,47834,110594,72761
C01131=-109333,-141938,-110765,47268,109335,72096
C01132=-106839,-147244,-109723,47050,105697,71521
C01133=-96955,-158208,-128899,-2670,111185,56030
C01134=-107130,-144670,-115956,-40497,90070,47196
C01135=-107133,-145289,-116877,-40503,90261,47122
C01136=-107139,-146938,-119316,-40521,90762,46927
C01137=-81304,-146505,-131302,-46256,99624,33732
C01138=-42290,-135810,-134986,-6789,56953,-43412
C01139=-53482,-111499,-99357,-5283,31563,-44884
C01140=-53488,-110753,-96932,-5448,30458,-44798
C01141=-53106,-110845,-96482,-5998,30161,-44520
C01142=-53143,-110117,-93832,-6189,28906,-44421
C01143=-53188,-109818,-93168,-6175,28651,-44427
C01144=-53095,-108922,-90553,-6542,27518,-44240
C01145=-53472,-108968,-91791,-5862,28222,-44586
C01146=-53466,-109889,-94290,-5675,29282,-44681
C01147=-93748,-113667,-111432,27227,62688,-41579
C01148=-93751,-113561,-109328,27520,61581,-41869
C01149=-94535,-110348,-107800,27711,62471,-41963
C01150=-94560,-109570,-102150,28499,59749,-42715
C01151=-93743,-112935,-104615,28181,59286,-42489
C01152=-93741,-113330,-106821,27872,60309,-42206
C01153=-53707,-103235,-126817,-3349,90409,-72793
C01154=-53694,-107630,-124107,-3352,86490,-72685
C01155=-53689,-108955,-122884,-3357,85060,-72645
C01156=-53697,-108940,-122873,-3354,85062,-72648
C01157=-53721,-108898,-122839,-3346,85062,-72656
C01158=-53729,-108884,-122827,-3345,85059,-72658
C01159=-53735,-107561,-124050,-3339,86489,-72698
C01160=-53748,-103173,-126762,-3336,90406,-72805
C01161=-44251,-68518,-112793,-6305,100072,-70363
C01162=-80270,30794,-42629,-11133,115571,-76543
C01163=-69737,67118,16632,-42575,112328,-80617
C01164=-69636,63823,22197,-49512,110599,-81416
C01165=-67564,55530,12856,-50142,112647,-81508
C01166=-66424,44944,1253,-49852,108764,-84350
C01167=-65618,29495,-14632,-48008,102670,-88237
C01168=-64581,15750,-27557,-48396,103780,-88326
C01169=-64160,11595,-31362,-48525,104124,-88308
C01170=-61878,-10748,-50140,-48981,105285,-87846
C01171=-62672,195,-41330,-51307,112408,-84907
C01172=-58944,10301,-35991,-52571,115494,-84879
C01173=-69716,-6230,-69222,-29298,97742,-75748
C01174=-102330,-22799,-82036,11222,88832,-73278
C01175=-48313,-118911,-129560,19207,92704,-27073
C01176=-53495,-110604,-121584,20154,93282,-28749
C01177=-53400,-112789,-120712,20093,91701,-28982
C01178=-53738,-109625,-119688,20178,92712,-28930
C01179=-53963,-109991,-119979,20218,92760,-28997
C01180=-54259,-112639,-122766,20278,93161,-29031
C01181=-53522,-108468,-123882,20258,95652,-28360
C01182=-66910,-101677,-117691,1645,82254,17515
C01183=-66905,-103395,-115374,1652,79946,17486
C01184=-66559,-103374,-114061,1536,79140,17588
C01185=-66525,-103141,-114029,1523,79241,17602
C01186=-67620,-103650,-114144,1902,79074,17240
C01187=-69811,-106122,-108316,12679,69437,17327
C01188=-66783,-105788,-110032,11324,70201,18483
C01189=-66785,-105108,-112553,11207,72068,18659
C01190=-34610,-119076,-126707,-31995,89279,47352
C01191=-26693,-119602,-105841,-51320,82883,62074
C01192=-26676,-118953,-103885,-51392,82336,62389
C01193=-26611,-118260,-103653,-51381,82509,62328
C01194=-26639,-116853,-99731,-51529,81413,62927
C01195=-26666,-118021,-101324,-51491,81640,62785
C01196=-26683,-118745,-103309,-51412,82173,62476
C01197=-26741,-121947,-116429,-51038,86269,60171
C01198=-80158,-111738,-121779,-46707,81282,-33331
C01199=-80124,-114295,-114082,-47454,77096,-31277
C01200=-80115,-114367,-110881,-47781,75720,-30584
C01201=-79768,-115533,-110081,-48056,75157,-30124
C01202=-79863,-115342,-112075,-47802,76014,-30606
C01203=-81971,-122337,-112055,-47997,72434,-29847
C01204=-79704,-115764,-110171,-48082,75146,-30085
C01205=-122148,-120937,-111499,-32844,53810,-41506
C01206=-126062,-118880,-110838,-30416,52910,-43086
C01207=-126117,-120875,-113087,-30250,53200,-43207
C01208=-80061,-114542,-114188,-47480,77086,-31241
C01209=-80063,-113108,-120040,-30435,104055,-77976
C01210=-80050,-114212,-116860,-30086,101864,-77373
C01211=-80380,-112077,-114717,-30053,101557,-77419
C01212=-79932,-114590,-112006,-35005,85347,-77215
C01213=-79912,-114566,-112044,-35008,85386,-77219
C01214=-80479,-112475,-109427,-36632,80098,-77307
C01215=-80029,-114714,-111597,-36713,80437,-77233
C01216=-82440,-93132,-104306,-35744,84828,-79668
C01217=-83378,-90315,-100640,-35536,83784,-79702
C01218=-86724,-76310,-94495,-34501,85296,-81493
C01219=-81341,-82881,-101909,-35963,88366,-80388
C01220=-80042,-114535,-115070,-36542,82240,-77847
C01221=-80040,-111621,-122742,-8414,85267,-41918
C01222=-80035,-113457,-119567,-8450,82400,-41723
C01223=-81798,-124774,-120168,-7328,73182,-41674
C01224=-80327,-109577,-118133,2572,87034,-53415
C01225=-79380,-112621,-119090,2349,86031,-53125
C01226=-78889,-114029,-118891,6085,83597,-58153
C01227=-80002,-113603,-119620,10752,83390,-63441
C01228=-80006,-103113,-128729,10775,94202,-62513
C01229=-39776,-103787,-110683,-21075,62663,59255
C01230=-39766,-104399,-107995,-21452,60825,59622
C01231=-41663,-99518,-106576,-17765,63773,58656
C01232=-39441,-104963,-106701,-21848,59898,59942
C01233=-39326,-105104,-106740,-21922,59881,59993
C01234=-39744,-104425,-108009,-21464,60826,59630
C01235=-39754,-103814,-110697,-21087,62664,59263
C01236=-47977,-106691,-119962,-23629,83327,62671
C01237=-66867,-99660,-121232,-22132,99220,62132
C01238=-66851,-102572,-118810,-21937,96446,62653
C01239=-74494,-137000,-128982,-14609,78071,53501
C01240=-72467,-138184,-128020,-15181,77278,54315
C01241=-67516,-140688,-126942,-16493,76361,56201
C01242=-43056,-127353,-114280,-36292,85121,62743
C01243=-66851,-103895,-117201,-21852,94891,62938
C01244=-66868,-101493,-119792,-22004,97521,62449
C01245=-74321,-107832,-126985,11736,80239,61811
C01246=-66584,-114412,-108983,34198,49386,64476
C01247=-66581,-113854,-105403,35147,47795,63826
C01248=-59001,-125725,-103773,32485,32454,61113
C01249=-65790,-113886,-101008,36132,45231,63145
C01250=-65568,-123466,-98279,45853,34675,56822
C01251=-65581,-123771,-97752,46366,34344,56544
C01252=-66567,-113311,-102857,35821,46729,63375
C01253=-66569,-114089,-106515,34851,48256,64025
C01254=-52763,-107501,-118592,5184,62268,61653
C01255=-39766,-104399,-107995,-21452,60825,59622
C01256=-42284,-99628,-106389,-17466,63479,58468
C01257=-39837,-104496,-106407,-21621,59851,59791
C01258=-39825,-104515,-106407,-21630,59842,59799
C01259=-39744,-104425,-108009,-21464,60826,59630
C01260=-39754,-103814,-110697,-21087,62664,59263
C01261=-47977,-106691,-119962,-23629,83327,62671
C01262=-66867,-99660,-121232,-22132,99220,62132
C01263=-66851,-102572,-118810,-21937,96446,62653
C01264=-75086,-136456,-128394,-14464,77886,53317
C01265=-72467,-138185,-128020,-15181,77278,54315
C01266=-67700,-141101,-127057,-16459,76187,56159
C01267=-43685,-128094,-114664,-36232,84741,62610
C01268=-66851,-103895,-117201,-21852,94891,62938
C01269=-66868,-101493,-119792,-22004,97521,62449
C01270=-74321,-107832,-126985,11736,80239,61811
C01271=-66584,-114412,-108983,34198,49386,64476
C01272=-66581,-113854,-105403,35147,47795,63826
C01273=-59470,-125293,-103644,32823,32756,60929
C01274=-65940,-113573,-100903,36174,45372,63123
C01275=-65237,-123018,-98144,45460,34612,57042
C01276=-65306,-123403,-97643,46040,34287,56728
C01277=-66567,-113311,-102857,35821,46729,63375
C01278=-66569,-114089,-106515,34851,48256,64025
C01279=-66614,-114312,-115902,32344,53032,65825
C01280=-26293,-124733,-123676,35115,86081,77095
C01281=-26278,-124914,-120130,35186,84196,76502
C01282=-26550,-125631,-118910,35285,83385,76132
C01283=-26140,-123752,-118256,35186,83681,76394
C01284=-26301,-124893,-120124,35190,84211,76498
C01285=-26317,-124710,-123669,35119,86096,77090
C01286=-26368,-124828,-121889,39154,95960,78120
C01287=-26350,-124746,-118556,38992,94373,77544
C01288=-26342,-124553,-116950,38932,93670,77290
C01289=-26340,-123995,-113991,38847,92461,76851
C01290=-26347,-124286,-115407,38884,93032,77056
C01291=-26365,-124761,-118865,39006,94524,77592
C01292=-26264,-124528,-116402,47920,86072,68134
C01293=-26249,-123768,-112787,47988,84810,67516
C01294=-26243,-123374,-111311,48022,84325,67278
C01295=-26226,-122772,-109280,48074,83674,66962
C01296=-26232,-123227,-110778,48035,84146,67194
C01297=-26247,-124165,-114452,47952,85370,67795
C01298=-82585,-123093,-118421,52491,64599,59558
C01299=-107155,-118824,-102398,58122,50036,52281
C01300=-107155,-117467,-98958,59145,49269,51564
C01301=-96813,-117817,-104188,42223,47347,50994
C01302=-105933,-121077,-109912,10415,42869,62990
C01303=-105953,-121074,-109843,10442,42831,62975
C01304=-107149,-121400,-109798,11502,42801,62375
C01305=-106717,-121349,-105974,7567,38238,71665
C01306=-107169,-120346,-107141,7797,39493,71540
C01307=-108433,-119625,-117514,7930,46308,71537
C01308=-107111,-122100,-111275,39348,45202,56077
C01309=-107109,-117760,-98763,43179,41028,53713
C01310=-106761,-117495,-97713,43363,40478,53604
C01311=-106458,-119074,-102370,12274,36991,61895
C01312=-105683,-116022,-101280,9396,37560,63477
C01313=-85991,-103596,-98751,-25015,50891,70344
C01314=-83847,-106333,-107319,-25140,55050,70229
C01315=-110745,-121766,-106380,43469,44759,53583
C01316=-110745,-121766,-106380,43469,44759,53584
C01317=-120731,-110814,-96413,59684,53172,46713
C01318=-94986,-115649,-101302,-12294,38121,75258
C01319=-110957,-117259,-94521,-45268,37979,76630
C01320=-107127,-114270,-91297,-56630,43098,80056
C01321=-102543,-110504,-99650,-53136,49996,77723
C01322=-93612,-109275,-133010,12113,75674,64968
C01323=-74458,-81913,-116300,25886,107898,47202
C01324=-74285,-84923,-113224,25351,104735,46539
C01325=-74085,-86300,-112083,25142,103399,46313
C01326=-71499,-76504,-108067,25490,106819,45523
C01327=-62961,-60085,-100217,24652,107848,48688
C01328=-60437,-59805,-99888,23461,105440,51393
C01329=-60588,-58283,-100875,23679,106756,51616
C01330=-60637,-54628,-103477,24231,109960,52288
C01331=-76657,-70403,-83915,51355,64349,40407
C01332=-74830,-68241,-74355,53953,55282,38932
C01333=-73110,-62379,-68708,53436,54020,39148
C01334=-73182,-62563,-68609,53555,53963,39058
C01335=-36930,-67607,-75173,-26029,44061,77403
C01336=-80523,-89058,-85253,18218,36719,55154
C01337=-82272,-90569,-85112,18702,34759,56728
C01338=-81508,-95500,-88175,18158,33969,56993
C01339=-81043,-103588,-94156,17854,33413,57140
C01340=-82846,-88179,-88219,41798,48730,43563
C01341=-81818,-81213,-82326,41198,48211,43888
C01342=-79663,-80074,-80946,37957,46333,45127
C01343=-64011,-84834,-85332,4259,39755,58703
C01344=-75846,-87347,-86370,15921,40584,52659
C01345=-47572,-67654,-78731,-37306,60592,66422
C01346=-46339,-68382,-80235,-37741,61555,66618
C01347=-42699,-70655,-83815,-39176,63943,67342
C01348=-43803,-67144,-92021,-36183,69839,64523
C01349=-86906,-70734,-117845,25978,101850,24881
C01350=-194376,-118372,-116958,36622,58194,-75254
C01351=-187943,-106127,-101715,33777,52366,-74665
C01352=-187951,-105693,-98645,34509,50978,-75202
C01353=-187954,-105458,-97394,34809,50440,-75417
C01354=-187960,-105469,-97402,34805,50444,-75420
C01355=-187927,-105629,-98482,19599,46235,-60273
C01356=-187923,-105820,-99644,19403,46817,-60144
C01357=-187914,-106157,-102495,18928,48312,-59826
C01358=-188021,-109107,-91072,54887,40419,-77132
C01359=-188025,-108188,-88773,55807,39869,-77674
C01360=-188027,-107805,-87846,56180,39654,-77892
C01361=-188036,-107761,-87717,56242,39627,-77928
C01362=-188035,-108145,-88644,55869,39841,-77710
C01363=-188030,-109068,-90945,54948,40390,-77168
C01364=-188015,-114130,-110744,41340,72657,-75143
C01365=-188018,-113864,-107763,41683,71368,-75679
C01366=-188019,-113684,-106544,41824,70871,-75888
C01367=-188009,-113674,-106577,41816,70886,-75877
C01368=-188008,-113852,-107795,41674,71383,-75668
C01369=-188005,-114114,-110775,41332,72673,-75132
C01370=-187933,-113872,-110928,18210,58720,-57176
C01371=-187882,-113256,-105308,-719,43762,-42538
C01372=-187896,-112711,-102669,-725,42418,-42533
C01373=-187852,-113170,-101841,-775,41671,-42505
C01374=-187778,-112374,-98354,-1639,37547,-42296
C01375=-187899,-111729,-99017,-1491,38283,-42378
C01376=-187886,-112431,-101600,-1465,39511,-42393
C01377=-192869,-127835,-120494,22551,66263,-53872
C01378=-188079,-122619,-114609,40714,83609,-61664
C01379=-188077,-122103,-112045,40794,82601,-62056
C01380=-188097,-121812,-110726,41966,87288,-59780
C01381=-188097,-121769,-110559,41966,87227,-59806
C01382=-188105,-121282,-108770,41980,86589,-60067
C01383=-188106,-121566,-109755,41972,86936,-59927
C01384=-188110,-122188,-112187,41960,87826,-59570
C01385=-188058,-121965,-125191,40549,88870,-59628
C01386=-104402,-90439,-123637,22599,88102,26907
C01387=-80407,-121901,-119741,18448,66455,46046
C01388=-99207,-113247,-119914,5586,82670,39005
C01389=-101996,-106609,-115785,6360,83734,38140
C01390=-119008,-118478,-113260,32340,76336,33375
C01391=-80488,-121328,-114439,18908,63658,45548
C01392=-79672,-120202,-114057,18494,63797,45891
C01393=-79592,-120276,-114079,18461,63755,45915
C01394=-80475,-121542,-115946,18779,64427,45684
C01395=-80482,-121578,-119613,18469,66554,46034
C01396=-85156,-144709,-129107,-21632,59402,64028
C01397=-93856,-120445,-109825,-39450,57641,70752
C01398=-93847,-119691,-106928,-40019,56559,71233
C01399=-86628,-99816,-98593,-45940,69277,74290
C01400=-86043,-99167,-98859,-45014,69635,74495
C01401=-83318,-93529,-94650,-47165,68336,75996
C01402=-93680,-116508,-100417,-40719,46210,72415
C01403=-93820,-118277,-102341,-40471,46353,72255
C01404=-93828,-119232,-105178,-39715,47322,71755
C01405=-93822,-120125,-107980,-28359,52237,38282
C01406=-93816,-119582,-106091,-28689,51458,38525
C01407=-93813,-119346,-105328,-28822,51152,38622
C01408=-93805,-118409,-102529,-29499,49391,39302
C01409=-93820,-119862,-107056,-29266,59584,40856
C01410=-93823,-120114,-107958,-29147,59957,40747
C01411=-93830,-120670,-110185,-28854,60909,40473
C01412=-63807,-119595,-131717,-32346,77391,31957
C01413=-66677,-121755,-125547,-9668,69981,-32239
C01414=-66675,-122709,-116301,-10101,63887,-31721
C01415=-66675,-122586,-115330,-10147,63360,-31673
C01416=-66678,-122782,-121307,9429,81851,-37654
C01417=-66765,-122962,-121469,9451,81867,-37681
C01418=-66675,-122328,-113778,33290,107246,-42961
C01419=-66675,-122499,-114776,33395,107690,-42822
C01420=-66677,-122795,-117228,33681,108831,-42458
C01421=-67830,-119002,-127241,35733,116022,-40496
C01422=-66677,-118144,-130351,-9432,74728,-32617
C01423=-66675,-122709,-116301,-10101,63887,-31721
C01424=-66675,-122566,-115195,-10154,63288,-31666
C01425=-66598,-122626,-121075,9408,81779,-37632
C01426=-62201,-135334,-124977,8438,77219,-36455
C01427=-72037,-126014,-118725,27283,91958,-49043
C01428=-76379,-123759,-128626,28058,99823,-48794
C01429=-71006,-123079,-126009,31798,108132,-44322
C01430=-66720,-122114,-124411,34847,112827,-41144
C01431=-125074,-112778,-121368,18538,134713,-61704
C01432=-173715,-145384,-131232,-10200,126221,-84589
C01433=-173715,-147046,-136936,-18176,117071,-78230
C01434=-173715,-145384,-131232,-55285,56270,-43989
C01435=-121435,-145384,-131232,-55285,56270,-43989
C01436=-118035,-115309,-97908,-59229,55500,-40903
C01437=-129283,-161545,-102403,-79044,40043,-30541
C01438=-116007,-110364,-98843,-57726,100679,-36272
C01439=-114404,-140880,-107972,-56001,95951,-32046
C01440=-114314,-138738,-101986,-58000,106431,-39451
C01441=-102008,-144788,-123359,-59173,119414,-41279
C01442=-15972,-110889,-128286,-10965,59905,-43045
C01443=-15972,-110889,-128286,-10965,59905,-43045
C01444=-101389,-60822,-75148,6919,68546,-70102
C01445=-115790,69230,64798,-8053,66131,-71909
C01446=-120688,105020,73307,-12402,84846,-73777
C01447=-120868,103639,75593,-12409,82749,-73629
C01448=-120940,103216,76680,-12418,81872,-73566
C01449=-120940,103732,79019,-12450,80724,-73451
C01450=-120940,103216,76680,-12418,81872,-73566
C01451=-120298,112004,89967,-12640,78393,-72988
C01452=-120707,106255,82361,-12511,80017,-73298
C01453=-120298,112004,89967,-12640,78393,-72988
C01454=-120298,111380,88066,-12608,79223,-73073
C01455=-122096,108036,83635,-12280,79933,-73777
C01456=-122096,108524,85355,-12307,79144,-73698
C01457=-121742,108481,85298,-12365,79210,-73582
C01458=-121911,108228,84384,-12322,79608,-73681
C01459=-120228,112105,88453,-12614,79365,-73063
C01460=-120053,112844,85327,-12571,81642,-73235
C01461=-120830,71540,61874,-4756,55589,-66514
C01462=-120535,76858,72419,-5134,51864,-66212
C01463=-120418,79487,77321,-5314,50212,-66075
C01464=-120418,81305,81326,-5435,48689,-65991
C01465=-120418,79487,77321,-5314,50212,-66075
C01466=-121101,73566,71896,-4942,50464,-66384
C01467=-120640,77942,77238,-5256,49458,-66131
C01468=-121101,73566,71896,-4942,50464,-66384
C01469=-121222,71175,67349,-4775,52021,-66512
C01470=-121527,66226,57370,-4418,55590,-66797
C01471=-120817,46858,51705,6808,46216,-80289
C01472=-120487,52530,62238,7041,42645,-80409
C01473=-120357,55197,66992,7170,41090,-80474
C01474=-120357,57219,71131,7393,39594,-80606
C01475=-120357,55197,66992,7170,41090,-80474
C01476=-121171,51687,64922,7778,40638,-80922
C01477=-120657,55397,69123,7546,39918,-80729
C01478=-121171,51687,64922,7778,40638,-80922
C01479=-121307,49062,60252,7635,42163,-80850
C01480=-121648,43436,49847,7373,45678,-80715
C01481=-109578,66950,51259,-9202,73878,-70224
C01482=-101389,-60822,-75148,6919,68546,-70102
C01483=-96929,-90691,-89138,5080,61517,-23019
C01484=-96929,-90691,-89138,5080,61517,27168
C01485=-133997,38575,-5386,4879,105902,64390
C01486=-134430,35731,-4221,4855,103756,64161
C01487=-134605,34666,-3678,4847,102887,64068
C01488=-134604,34193,-2477,4825,101908,64030
C01489=-134605,34666,-3678,4847,102887,64068
C01490=-133324,38381,1851,4717,101326,64430
C01491=-133984,36157,-436,4773,101627,64224
C01492=-133324,38381,1851,4717,101326,64430
C01493=-132740,42105,45,4739,104308,64739
C01494=-159526,23962,790,32225,80504,55500
C01495=-158922,24925,5721,32299,78113,55050
C01496=-158153,25889,7618,32183,77247,55110
C01497=-158153,25992,9261,32290,76429,54873
C01498=-158153,25975,9034,32275,76541,54905
C01499=-159336,23803,6937,32538,77140,54603
C01500=-159336,23824,7234,32557,76994,54560
C01501=-158542,24868,8237,32379,76622,54771
C01502=-158626,24722,8098,32398,76663,54749
C01503=-158626,24746,8414,32418,76509,54705
C01504=-158626,24723,8130,32399,76648,54745
C01505=-159596,23128,6599,32614,77122,54493
C01506=-159596,23153,6932,32637,76960,54446
C01507=-159062,24432,8187,32525,76656,54571
C01508=-159244,23446,6313,32496,77274,54679
C01509=-160967,21427,101,32642,80299,54873
C01510=-147551,27169,-6215,28445,81493,60312
C01511=-147017,27605,-1759,28452,79091,59917
C01512=-146493,28433,829,28390,77886,59816
C01513=-146493,28355,1445,28429,77515,59723
C01514=-146493,28387,1187,28413,77670,59762
C01515=-147642,25561,-1571,28744,78267,59478
C01516=-147642,25516,-1231,28765,78061,59427
C01517=-146933,27046,255,28560,77712,59607
C01518=-147010,26749,-33,28581,77761,59589
C01519=-147010,26722,196,28596,77625,59555
C01520=-147010,26770,-196,28572,77860,59614
C01521=-147964,24407,-2486,28847,78350,59377
C01522=-147964,24325,-1833,28887,77960,59278
C01523=-147292,26053,-161,28694,77611,59445
C01524=-147523,24411,-2449,28713,78186,59502
C01525=-149162,23542,-7999,28991,81344,59682
C01526=-129846,-17397,-52274,16165,101048,68229
C01527=-103949,-6271,-30701,7884,96105,76175
C01528=-94102,16895,-5866,4380,94047,79161
C01529=-94024,14878,-3719,4358,91692,79105
C01530=-93993,14152,-2780,4351,90742,79083
C01531=-93993,14213,-1554,4335,90021,79057
C01532=-93993,14202,-1750,4335,90136,79060
C01533=-93544,18458,2169,4295,89888,79203
C01534=-93544,18476,2442,4295,89728,79198
C01535=-93713,17041,1146,4310,89799,79144
C01536=-93671,17336,1418,4307,89780,79158
C01537=-93671,17356,1712,4307,89607,79151
C01538=-93671,17342,1501,4307,89730,79155
C01539=-93486,20302,4269,4303,89540,79209
C01540=-93873,20584,4779,4336,89392,79073
C01541=-94001,18334,2673,4347,89541,79036
C01542=-94106,19042,2519,4357,90004,79017
C01543=-93796,22544,1176,4343,92603,79213
C01544=-95224,-25687,-42365,27028,60157,72238
C01545=-94111,-23276,-36997,26973,57954,72128
C01546=-93597,-19509,-33603,26734,57655,72271
C01547=-93597,-19504,-31914,27029,56727,72023
C01548=-93597,-19510,-32243,26972,56905,72072
C01549=-93990,-24549,-35870,27293,56712,71846
C01550=-93990,-24538,-35459,27369,56492,71783
C01551=-93788,-21252,-33109,27186,56644,71914
C01552=-93840,-21553,-33328,27220,56642,71889
C01553=-93840,-21543,-33005,27278,56468,71842
C01554=-93840,-21553,-33351,27216,56655,71894
C01555=-94357,-24968,-35787,27577,56595,71647
C01556=-94357,-24947,-35259,27673,56314,71569
C01557=-94013,-22711,-33670,27433,56354,71733
C01558=-93814,-23881,-35617,27147,56823,71950
C01559=-95768,-30118,-43626,27714,58991,71694
C01560=-97625,-41604,-59467,17173,89706,-8843
C01561=-96114,-37688,-53918,16886,88057,-8555
C01562=-95526,-36022,-51615,16777,87400,-8443
C01563=-95527,-36150,-50037,16784,86406,-8579
C01564=-95526,-36022,-51615,16777,87400,-8443
C01565=-95532,-36183,-50637,16782,86745,-8534
C01566=-95234,-33170,-48668,16723,87008,-8396
C01567=-95532,-36183,-50637,16782,86745,-8534
C01568=-95504,-36095,-50208,16778,86530,-8554
C01569=-93996,-36675,-50581,16493,86163,-8084
C01570=-95504,-36095,-50208,16778,86530,-8554
C01571=-97625,-41604,-59467,17173,89706,-8843
C01572=-101873,-77751,-87156,42969,63075,62474
C01573=-95937,-74809,-81328,40948,58735,63434
C01574=-95565,-74583,-80935,40815,58468,63500
C01575=-95566,-74620,-79294,41227,57681,63141
C01576=-95565,-74583,-80935,40815,58468,63500
C01577=-98755,-73227,-80296,42221,60183,62682
C01578=-98803,-73638,-78797,42678,59356,62269
C01579=-96868,-74481,-79195,41849,58298,62761
C01580=-98803,-73638,-78797,42678,59356,62269
C01581=-97163,-69666,-76891,41573,59236,63045
C01582=-96752,-66139,-75134,41097,59602,63417
C01583=-97163,-69666,-76891,41573,59236,63045
C01584=-101873,-77751,-87156,42969,63075,62474
C01585=-126113,-49786,-51573,51544,90004,55144
C01586=-123973,-50127,-48217,51392,87374,54806
C01587=-123286,-49758,-46380,51349,86473,54664
C01588=-118478,-34750,-37348,50925,85086,56432
C01589=-119272,-35479,-39244,50973,86038,56539
C01590=-121232,-35158,-42579,51146,88553,56901
C01591=-111145,-57425,-62081,41633,61582,55088
C01592=-109620,-53993,-56645,41578,59663,54986
C01593=-109014,-52418,-54338,41560,58914,54950
C01594=-105531,-54881,-55720,40219,56972,55856
C01595=-106107,-56401,-57979,40230,57706,55889
C01596=-107578,-60042,-63488,40293,59558,55964
C01597=-93331,-25535,-46307,22677,87971,72102
C01598=-84242,-5399,-27465,11713,100257,81196
C01599=-83743,-8192,-25851,11599,97806,81134
C01600=-83603,-8644,-24372,11558,96668,81075
C01601=-80847,-8673,-24279,11462,96208,81977
C01602=-80973,-8366,-25985,11504,97411,82047
C01603=-81511,-5615,-27635,11617,99868,82095
C01604=-103949,-6271,-30701,7884,96105,76175
C01605=-129846,-17397,-52274,16165,101048,68229
C01606=-175693,57260,35469,48998,74273,48315
C01607=-174652,59964,42108,49342,71909,47593
C01608=-173879,58726,41837,48629,68835,47243
C01609=-174989,71180,56287,49602,67767,46055
C01610=-173482,53917,36869,46602,62532,46609
C01611=-174364,49990,29079,45939,64941,47387
C01612=-163099,39792,11105,47007,80916,54866
C01613=-161954,40669,15666,46993,78691,54338
C01614=-161544,42106,18156,47002,77926,54165
C01615=-160409,36094,11923,46622,77862,54687
C01616=-160850,34862,9687,46632,78611,54832
C01617=-162019,34035,5199,46665,80839,55343
C01618=-147988,42797,109,12455,106225,61454
C01619=-148219,40121,1423,12320,104123,61157
C01620=-146030,57026,21700,8846,110028,61895
C01621=-145258,50191,13883,9166,109401,62129
C01622=-144531,51862,16039,8885,111237,62498
C01623=-146794,35355,-3496,12271,104485,61677
C01624=-146567,38090,-4821,12411,106625,61976
C01625=-96929,-90691,-89138,5080,61517,27168
C01626=-96929,-90691,-89138,5080,61517,-23019
C01627=-101389,-60822,-75148,6919,68546,-70102
C01628=-109578,66950,51259,-9202,73878,-70224
C01629=-119285,73548,61078,-7759,54489,-67872
C01630=-119140,78931,71700,-8230,50768,-67516
C01631=-119018,68322,64494,-9513,43413,-66753
C01632=-123077,79861,78861,-6886,39527,-68452
C01633=-122308,90513,86215,-6785,47517,-68668
C01634=-122473,83260,72935,-6271,51921,-69036
C01635=-119074,82203,59752,-14757,75142,-72556
C01636=-112473,77653,55392,-16315,76732,-70397
C01637=-111583,66581,50085,-22599,68947,-68307
C01638=-112205,67748,51306,-22435,68636,-68485
C01639=-112809,96137,83372,-20713,72479,-69433
C01640=-121067,113951,104217,-8230,68834,-71393
C01641=-120880,99674,85606,-8530,71491,-71499
C01642=-121360,95237,80258,-8447,70766,-71619
C01643=-121396,72779,51526,-8459,68942,-71502
C01644=-134157,70152,49704,15847,72235,-43808
C01645=-133722,73949,59265,16087,68355,-44178
C01646=-133862,75249,62165,16247,67307,-44381
C01647=-129675,65866,51066,4701,64817,-31992
C01648=-128682,62362,47014,4314,65455,-31601
C01649=-130205,57581,36634,4742,69462,-32000
C01650=-130312,54578,33992,4779,69550,-32035
C01651=-129992,46081,35923,20239,67004,8502
C01652=-121496,43425,36833,5893,59088,22773
C01653=-120237,47252,43120,2387,56768,25932
C01654=-119972,47626,45454,2298,55515,26011
C01655=-128073,50557,47782,20949,62737,7811
C01656=-127834,53853,52717,21124,61417,7650
C01657=-123180,48310,46556,9691,56439,19302
C01658=-122651,35401,27095,8965,61652,19959
C01659=-109578,66950,51259,-9202,73878,-70224
C01660=-101389,-60822,-75148,6919,68546,-70102
C01661=-96929,-90691,-89138,5080,61517,-23019
C01662=-93242,-109726,-96296,3420,55961,28393
C01663=-92156,-22649,-39625,10516,94476,60392
C01664=-92890,-21952,-35043,10540,92147,59946
C01665=-92918,-23039,-34191,10529,91084,59847
C01666=-95371,-22229,-33611,10738,91463,59044
C01667=-94898,-22950,-35761,10710,92338,59280
C01668=-94492,-21797,-39017,10723,94837,59633
C01669=-92575,-26977,-42679,21088,73618,56030
C01670=-92430,-25186,-37423,21282,71416,55682
C01671=-92215,-23603,-34702,21309,70555,55605
C01672=-95579,-22098,-33596,23466,71740,54512
C01673=-95477,-23933,-36320,23344,72386,54682
C01674=-95719,-25683,-41558,23174,74597,55037
C01675=-96929,-90691,-89138,5080,61517,27168
C01676=-96929,-90691,-89138,5080,61517,-23019
C01677=-101389,-60822,-75148,6919,68546,-70102
C01678=-109578,66950,51259,-9202,73878,-70224
C01679=-108278,48890,46404,-6655,48460,-73563
C01680=-108252,54023,56228,-7048,45078,-73302
C01681=-107661,40825,52409,-14308,28668,-70428
C01682=-112610,50539,61242,-7713,29705,-74042
C01683=-112702,61866,65174,-4315,43297,-75310
C01684=-112766,56024,54314,-4011,46966,-75508
C01685=-103921,32533,46603,10708,30188,-75698
C01686=-104692,35200,60863,30413,16065,-83251
C01687=-104796,38679,66061,33302,14894,-84599
C01688=-102333,36267,63497,27606,14351,-81669
C01689=-100412,37194,55383,7603,26828,-73795
C01690=-100998,29868,43914,7479,30147,-73786
C01691=-109578,66950,51259,-9202,73878,-70224
C01692=-101389,-60822,-75148,6919,68546,-70102
C01693=-96929,-90691,-89138,5080,61517,-23019
C01694=-96929,-90691,-89138,5080,61517,27168
C01695=-90570,-23240,-39845,-1682,91658,61068
C01696=-90349,-1837,-19216,-4288,101242,62233
C01697=-91056,3798,-12678,-2790,103655,62048
C01698=-91511,6444,-9862,-6335,104149,61595
C01699=-95291,-22836,-35623,-1093,89189,59526
C01700=-94239,-22001,-38963,-1226,91687,59852
C01701=-90424,-29050,-43505,3763,58999,61302
C01702=-86008,-21130,-36360,-6353,62529,61992
C01703=-86318,-18191,-32565,-6237,61686,61924
C01704=-89142,-17607,-32133,-4748,61529,60871
C01705=-95351,-24457,-36663,6763,57473,59317
C01706=-94707,-27619,-42528,6252,59394,59681
C01707=-109011,-26713,-50438,8452,98222,74634
C01708=-144543,31549,-11380,-159,92982,60584
C01709=-143093,45679,4448,-4866,97184,60249
C01710=-142229,53785,16152,-6705,99618,60162
C01711=-144891,70831,35748,-7385,98802,59208
C01712=-148937,42537,3991,922,89189,59187
C01713=-148250,43318,770,754,91565,59420
C01714=-172279,3947,-14828,46151,77384,48319
C01715=-167570,-10636,-17777,41693,62852,42800
C01716=-166476,-7066,-11974,41907,61016,42522
C01717=-168831,4679,-2271,42697,62201,41872
C01718=-172859,17944,7820,47479,72977,45875
C01719=-174013,15583,1984,47261,75226,46421
C01720=-109011,-26713,-50438,8452,98222,74634
C01721=-99312,-50897,-61026,22837,72179,74454
C01722=-98138,-49989,-56545,22703,69739,74412
C01723=-106382,-52347,-50887,37007,65807,70627
C01724=-98813,-18962,-39289,22939,92751,75811
C01725=-101547,-27333,-44313,25543,91651,74875
C01726=-97857,-18198,-39852,20610,99055,76884
C01727=-96922,-25876,-47272,18742,95048,76352
C01728=-97638,-23312,-49453,18962,97729,76524
C01729=-81141,-50558,-66105,12803,46081,75388
C01730=-80687,-46119,-60183,12697,44679,75401
C01731=-80513,-44339,-57785,12667,44105,75401
C01732=-80516,-44488,-54802,13120,42239,75121
C01733=-80690,-46329,-57233,13145,42803,75122
C01734=-81145,-50923,-63237,13239,44177,75109
C01735=-83601,15534,-39616,9664,96262,77072
C01736=-80484,90945,50155,4324,118905,78550
C01737=-80490,84570,45509,4303,118490,78531
C01738=-80493,82108,43801,4293,118276,78521
C01739=-80495,81630,46278,4216,116511,78452
C01740=-80492,84058,47940,4226,116735,78462
C01741=-83493,53381,-2692,9637,111099,78940
C01742=-91945,-14209,-43630,9790,83010,75128
C01743=-10907,-117335,-90652,-18762,63715,-59495
C01744=-15972,-110889,-128286,-10965,59905,-43045
BC00000=48829,688840,1075175
BC00001=366911,902233,1075175
BC00002=366911,902233,1075175
BC00003=366911,902233,1075175
BC00004=366911,902233,1075175
BC00005=366911,902233,1075175
BC00006=366911,902233,1075175
BC00007=366911,902233,1075175
BC00008=366911,902233,1075175
BC00009=333056,895412,1075175
BC00010=333056,895412,1075175
BC00011=333056,895412,1075175
BC00012=333056,895412,1075175
BC00013=333056,895412,1075175
BC00014=333056,895412,1075175
BC00015=333056,895412,1075175
BC00016=333056,895412,1075175
BC00017=358091,902222,1075175
BC00018=358091,902222,1075175
BC00019=358091,902222,1075175
BC00020=358091,902222,1075175
BC00021=358091,902222,1075175
BC00022=358091,902222,1075175
BC00023=358091,902222,1075175
BC00024=358091,902222,1075175
BC00025=398174,894103,1075175
BC00026=398174,894103,1075175
BC00027=398174,894103,1075175
BC00028=398174,894103,1075175
BC00029=398174,894103,1075175
BC00030=398174,894103,1075175
BC00031=398174,894103,1075175
BC00032=398174,894103,1075175
BC00033=264903,781270,1075175
BC00034=264903,781270,1075175
BC00035=264904,781269,1075172
BC00036=264904,781269,1075171
BC00037=264904,781269,1075171
BC00038=264904,781269,1075168
BC00039=264904,781269,1075168
BC00040=264904,781269,1075168
BC00041=264904,781269,1075168
BC00042=264904,781269,1075168
BC00043=264904,781269,1075164
BC00044=264903,781270,1075175
BC00045=301264,775814,1075175
BC00046=301264,775814,1075175
BC00047=301264,775814,1075175
BC00048=301264,775814,1075175
BC00049=301264,775814,1075175
BC00050=301264,775814,1075175
BC00051=301264,775814,1075175
BC00052=301264,775814,1075175
BC00053=301264,775814,1075175
BC00054=301264,775814,1075175
BC00055=274235,786209,1075175
BC00056=238672,799885,1075175
BC00057=238672,799885,1075175
BC00058=238672,799885,1075175
BC00059=238672,799885,1075175
BC00060=238672,799885,1075175
BC00061=238672,799885,1075175
BC00062=238672,799885,1075175
BC00063=238672,799885,1075175
BC00064=238672,799884,1075171
BC00065=238672,799884,1075171
BC00066=238672,799885,1075175
BC00067=238672,799885,1075175
BC00068=238672,799885,1075175
BC00069=238672,799885,1075175
BC00070=318263,750454,1075175
BC00071=318263,750454,1075175
BC00072=318263,750454,1075175
BC00073=318263,750454,1075175
BC00074=318263,750454,1075175
BC00075=318263,750454,1075175
BC00076=318263,750454,1075175
BC00077=318263,750454,1075175
BC00078=318263,750454,1075175
BC00079=318263,750454,1075175
BC00080=318263,750454,1075175
BC00081=318263,750454,1075175
BC00082=318263,750454,1075175
BC00083=318263,750454,1075175
BC00084=318263,750454,1075175
BC00085=318263,750454,1075175
BC00086=318263,750454,1075175
BC00087=318263,750454,1075175
BC00088=318263,750454,1075175
BC00089=318263,750454,1075175
BC00090=318263,750454,1075175
BC00091=318263,750454,1075175
BC00092=318263,750454,1075175
BC00093=318263,750454,1075175
BC00094=318263,750454,1075175
BC00095=377114,750454,1075175
BC00096=397814,750454,1075175
BC00097=397814,750454,1075175
BC00098=397814,750454,1075175
BC00099=397814,750454,1075175
BC00100=397814,750454,1075175
BC00101=397814,750454,1075175
BC00102=397814,750454,1075175
BC00103=397814,750454,1075175
BC00104=397814,750454,1075175
BC00105=397814,750454,1075175
BC00106=397814,750454,1075175
BC00107=397814,750454,1075175
BC00108=397814,750454,1075175
BC00109=397814,750454,1075175
BC00110=397814,750454,1075175
BC00111=397814,750454,1075175
BC00112=397814,750454,1075175
BC00113=397814,750454,1075175
BC00114=397814,750454,1075175
BC00115=397814,750454,1075175
BC00116=383090,762961,1075175
BC00117=372387,772052,1075175
BC00118=296274,836703,1075175
BC00119=296274,836703,1075175
BC00120=296274,836703,1075175
BC00121=296274,836703,1075175
BC00122=296274,836703,1075175
BC00123=296274,836703,1075175
BC00124=296274,836703,1075175
BC00125=296274,836703,1075175
BC00126=296274,836703,1075175
BC00127=296274,836703,1075175
BC00128=296274,836703,1075175
BC00129=296274,836703,1075175
BC00130=296274,836703,1075175
BC00131=312215,899988,1075175
BC00132=312215,944285,1075175
BC00133=312215,944285,1075175
BC00134=312215,944285,1075175
BC00135=312215,944285,1075175
BC00136=312215,944285,1075175
BC00137=312215,944285,1075175
BC00138=312215,944285,1075175
BC00139=312215,944285,1075175
BC00140=312215,944285,1075175
BC00141=312215,944285,1075175
BC00142=312215,944285,1075175
BC00143=259299,938961,1075175
BC00144=259299,938961,1075175
BC00145=259299,938961,1075175
BC00146=259299,938961,1075175
BC00147=259299,938961,1075175
BC00148=259299,938961,1075175
BC00149=259299,938961,1075175
BC00150=259299,938961,1075175
BC00151=259299,938961,1075175
BC00152=259299,938961,1075175
BC00153=259299,938961,1075175
BC00154=259299,938961,1075175
BC00155=211531,951911,1075175
BC00156=211531,951911,1075175
BC00157=211531,951911,1075175
BC00158=211531,951911,1075175
BC00159=211531,951911,1075175
BC00160=211531,951911,1075175
BC00161=211531,951911,1075175
BC00162=211531,951911,1075175
BC00163=211531,951911,1075175
BC00164=211531,951911,1075175
BC00165=211531,951911,1075175
BC00166=182503,951872,1075175
BC00167=184369,953383,1075175
BC00168=184369,953399,1075175
BC00169=184333,953526,1075175
BC00170=184897,956550,1075175
BC00171=184333,953526,1075175
BC00172=184751,953664,1075175
BC00173=187887,953121,1075175
BC00174=184751,953664,1075175
BC00175=178222,948378,1075175
BC00176=185204,949959,1075175
BC00177=186100,954799,1075175
BC00178=186458,956743,1075174
BC00179=186459,956752,1075175
BC00180=186578,956775,1075175
BC00181=187141,959799,1075175
BC00182=186578,956775,1075175
BC00183=185324,949999,1075175
BC00184=153081,998123,1075175
BC00185=123088,1061215,1075175
BC00186=126332,1055781,1075175
BC00187=127630,1053613,1075175
BC00188=127630,1053623,1075175
BC00189=127630,1053607,1075175
BC00190=153753,1064749,1075175
BC00191=152152,1062093,1075175
BC00192=153753,1064749,1075175
BC00193=104366,1038154,1075175
BC00194=107120,1036610,1075175
BC00195=104366,1038154,1075175
BC00196=97490,1044180,1075175
BC00197=140343,1045718,1075175
BC00198=158643,1046375,1075175
BC00199=155464,1041036,1075175
BC00200=155106,1040455,1075175
BC00201=155106,1040463,1075175
BC00202=155288,1040367,1075175
BC00203=153687,1037711,1075175
BC00204=155288,1040367,1075175
BC00205=158891,1046297,1075175
BC00206=211337,993614,1075175
BC00207=274623,983932,1075175
BC00208=371761,1043051,1075175
BC00209=371761,1043051,1075175
BC00210=371761,1043051,1075175
BC00211=371761,1043051,1075175
BC00212=371761,1043051,1075175
BC00213=371761,1043051,1075175
BC00214=371761,1043051,1075175
BC00215=371761,1043051,1075175
BC00216=371761,1043051,1075175
BC00217=371761,1043051,1075175
BC00218=371761,1043051,1075175
BC00219=371761,1043051,1075175
BC00220=371761,1043051,1075175
BC00221=371761,1043051,1075175
BC00222=371761,1043051,1075175
BC00223=314185,938855,1075175
BC00224=247671,970611,1075175
BC00225=247671,970611,1075175
BC00226=247671,970611,1075175
BC00227=247671,970611,1075175
BC00228=247671,970611,1075175
BC00229=247671,970611,1075175
BC00230=247671,970611,1075175
BC00231=247671,970611,1075175
BC00232=247671,970611,1075175
BC00233=247671,970611,1075175
BC00234=247671,970611,1075175
BC00235=247671,970611,1075175
BC00236=303037,872055,1075175
BC00237=380992,820655,1075175
BC00238=380992,820655,1075175
BC00239=380992,820655,1075175
BC00240=380992,820655,1075175
BC00241=380992,820655,1075175
BC00242=380992,820655,1075175
BC00243=380992,820655,1075175
BC00244=380992,820655,1075175
BC00245=380992,820655,1075175
BC00246=380992,820655,1075175
BC00247=380992,820655,1075175
BC00248=380992,820655,1075175
BC00249=275256,812324,1075175
BC00250=125716,897903,1075175
BC00251=125716,897903,1075175
BC00252=125716,897903,1075175
BC00253=125716,897903,1075175
BC00254=125716,897903,1075175
BC00255=125716,897903,1075174
BC00256=125716,897903,1075171
BC00257=125716,897903,1075175
BC00258=125716,897903,1075175
BC00259=125716,897903,1075175
BC00260=125716,897903,1075175
BC00261=125716,897903,1075175
BC00262=125716,897903,1075175
BC00263=325019,822543,1075229
BC00264=325019,822543,1075229
BC00265=325019,822543,1075229
BC00266=325019,822543,1075229
BC00267=325019,822543,1075229
BC00268=325019,822543,1075229
BC00269=325019,822543,1075229
BC00270=325019,822543,1075229
BC00271=325019,822543,1075229
BC00272=325019,822543,1075229
BC00273=325019,822543,1075229
BC00274=325019,822543,1075229
BC00275=240667,871930,1075210
BC00276=81335,965219,1075175
BC00277=81335,965219,1075175
BC00278=81335,965219,1075175
BC00279=81335,965219,1075175
BC00280=81335,965219,1075175
BC00281=81335,965219,1075175
BC00282=81335,965219,1075175
BC00283=81335,965219,1075175
BC00284=39891,972466,1075175
BC00285=39891,972466,1075175
BC00286=39891,972466,1075175
BC00287=39891,972466,1075175
BC00288=39891,972466,1075175
BC00289=39891,972466,1075175
BC00290=39891,972466,1075175
BC00291=39891,972466,1075175
BC00292=126064,942124,1075175
BC00293=145718,951183,1075175
BC00294=145718,951183,1075175
BC00295=145718,951183,1075175
BC00296=145718,951183,1075175
BC00297=145718,951183,1075175
BC00298=145718,951183,1075175
BC00299=145718,951183,1075175
BC00300=145718,951183,1075175
BC00301=145718,951183,1075175
BC00302=145718,951183,1075175
BC00303=145718,951183,1075175
BC00304=145718,951183,1075175
BC00305=127193,914007,1075175
BC00306=75497,867475,1075175
BC00307=75497,867475,1075175
BC00308=75497,867475,1075175
BC00309=75497,867475,1075175
BC00310=75497,867475,1075175
BC00311=75497,867475,1075175
BC00312=75497,867475,1075175
BC00313=75497,867475,1075175
BC00314=75497,867475,1075175
BC00315=75497,867475,1075175
BC00316=75497,867475,1075175
BC00317=75497,867475,1075175
BC00318=75497,867475,1075175
BC00319=75497,867475,1075175
BC00320=75497,867475,1075175
BC00321=75497,867475,1075175
BC00322=75497,867475,1075175
BC00323=58830,852413,1075175
BC00324=43274,838354,1075175
BC00325=43274,838354,1075175
BC00326=43274,838354,1075175
BC00327=43274,838354,1075175
BC00328=43274,838354,1075175
BC00329=43274,838354,1075175
BC00330=43274,838354,1075175
BC00331=43274,838354,1075175
BC00332=43274,838354,1075175
BC00333=191439,896290,1075175
BC00334=209593,874493,1075175
BC00335=209593,874493,1075175
BC00336=209593,874493,1075175
BC00337=209593,874493,1075171
BC00338=209593,874493,1075175
BC00339=209593,874493,1075175
BC00340=209216,850926,1075175
BC00341=226866,854473,1075175
BC00342=228835,855864,1075175
BC00343=228835,855864,1075175
BC00344=228834,855864,1075173
BC00345=228834,855864,1075173
BC00346=228835,855864,1075175
BC00347=228835,855864,1075175
BC00348=228835,855864,1075175
BC00349=228835,855864,1075175
BC00350=228835,855864,1075175
BC00351=212683,986357,1075175
BC00352=212683,1004517,1075175
BC00353=212247,999872,1075175
BC00354=212146,998778,1075171
BC00355=214955,996593,1075174
BC00356=222186,994128,1075175
BC00357=222622,998773,1075175
BC00358=293477,973063,1075175
BC00359=293477,973063,1075175
BC00360=293477,973063,1075175
BC00361=293477,973063,1075175
BC00362=293477,973063,1075175
BC00363=293477,973063,1075175
BC00364=293477,973063,1075175
BC00365=293477,973063,1075175
BC00366=248777,974412,1075175
BC00367=147624,1017934,1075175
BC00368=124950,1033375,1075175
BC00369=124950,1033375,1075175
BC00370=124950,1033375,1075175
BC00371=124950,1033375,1075175
BC00372=124950,1033375,1075175
BC00373=124950,1033375,1075175
BC00374=106678,1046165,1075175
BC00375=106678,1046165,1075175
BC00376=106678,1046165,1075175
BC00377=106678,1046165,1075175
BC00378=106678,1046165,1075175
BC00379=106678,1046165,1075175
BC00380=106678,1034404,1075175
BC00381=288363,951317,1075175
BC00382=319880,932288,1075175
BC00383=316203,930177,1075175
BC00384=314732,929332,1075175
BC00385=314732,929332,1075175
BC00386=294141,940882,1075175
BC00387=285351,949486,1075175
BC00388=280844,953897,1075175
BC00389=254356,968931,1075172
BC00390=253996,970793,1075175
BC00391=256777,973747,1075175
BC00392=224914,994659,1075175
BC00393=193407,1014756,1075175
BC00394=196552,1009267,1075175
BC00395=197065,1008372,1075175
BC00396=197397,1007797,1075175
BC00397=196552,1009278,1075175
BC00398=193407,1014766,1075175
BC00399=170876,1031134,1075175
BC00400=153007,1044116,1075175
BC00401=153007,1044116,1075175
BC00402=155599,1038213,1075175
BC00403=156636,1035851,1075175
BC00404=230598,1025728,1075175
BC00405=176896,1055708,1075175
BC00406=225377,1010635,1075175
BC00407=228184,1010601,1075175
BC00408=235201,1010515,1075175
BC00409=242597,980334,1075175
BC00410=282680,816770,1075175
BC00411=287393,774165,1075175
BC00412=293866,776192,1075175
BC00413=296455,777002,1075175
BC00414=296337,777088,1075175
BC00415=296308,777110,1075175
BC00416=296189,777197,1075175
BC00417=293600,776386,1075175
BC00418=287127,774359,1075175
BC00419=265173,805126,1075175
BC00420=271841,806848,1075175
BC00421=274508,807537,1075175
BC00422=274508,807537,1075175
BC00423=271842,806893,1075175
BC00424=265174,805171,1075175
BC00425=347775,809657,1075175
BC00426=348436,809459,1075175
BC00427=348700,809380,1075175
BC00428=352833,807067,1075175
BC00429=364813,800347,1075175
BC00430=368942,798027,1075175
BC00431=368677,798106,1075175
BC00432=368016,798304,1075175
BC00433=368016,798304,1075175
BC00434=391344,687000,1075175
BC00435=391344,687000,1075175
BC00436=391344,687000,1075175
BC00437=391344,687000,1075175
BC00438=391344,687000,1075175
BC00439=391344,687000,1075175
BC00440=391344,687000,1075175
BC00441=391344,687000,1075175
BC00442=391344,687000,1075175
BC00443=391344,687000,1075175
BC00444=391344,687000,1075175
BC00445=391344,687000,1075175
BC00446=358873,687000,1075175
BC00447=250171,896024,1075175
BC00448=255370,893912,1075175
BC00449=257449,893067,1075175
BC00450=259851,897051,1075175
BC00451=270502,914711,1075175
BC00452=268422,915555,1075175
BC00453=263223,917668,1075175
BC00454=251695,824506,1075175
BC00455=253916,829548,1075175
BC00456=254804,831565,1075175
BC00457=231448,844598,1075175
BC00458=231448,844598,1075175
BC00459=189878,862044,1075175
BC00460=188570,860127,1075175
BC00461=185301,855336,1075175
BC00462=261332,833542,1075175
BC00463=297112,823286,1075175
BC00464=293523,829343,1075175
BC00465=292087,831765,1075175
BC00466=292088,831788,1075175
BC00467=293523,829365,1075175
BC00468=297112,823308,1075175
BC00469=297112,823286,1075175
BC00470=112345,954746,1075175
BC00471=112345,954746,1075175
BC00472=111546,959512,1075175
BC00473=111226,961418,1075175
BC00474=63698,969650,1075175
BC00475=64018,967744,1075175
BC00476=64817,962978,1075175
BC00477=55529,859309,1075175
BC00478=51595,858048,1075175
BC00479=50021,857544,1075175
BC00480=45895,833192,1075175
BC00481=46071,849801,1075175
BC00482=43912,844296,1075175
BC00483=45475,843733,1075175
BC00484=45475,843733,1075175
BC00485=45475,843733,1075175
BC00486=45475,843733,1075175
BC00487=45475,843733,1075175
BC00488=49382,842326,1075175
BC00489=32191,855540,1075175
BC00490=35199,856902,1075175
BC00491=36402,857447,1075175
BC00492=24170,872455,1075175
BC00493=24116,855865,1075175
BC00494=17601,856883,1075175
BC00495=10106,858388,1075175
BC00496=7107,859694,1075175
BC00497=124165,958731,1075175
BC00498=124477,964204,1075175
BC00499=124602,966393,1075175
BC00500=119899,967208,1075175
BC00501=114659,968116,1075175
BC00502=114534,965927,1075175
BC00503=114222,960453,1075175
BC00504=169497,963360,1075175
BC00505=218455,965934,1075175
BC00506=214431,967961,1075175
BC00507=212822,968772,1075175
BC00508=212822,968772,1075175
BC00509=212822,968772,1075175
BC00510=212822,968772,1075175
BC00511=218344,963319,1075175
BC00512=222368,961291,1075175
BC00513=147324,958268,1075175
BC00514=86350,984014,1075175
BC00515=90717,985390,1075175
BC00516=92241,985755,1075175
BC00517=87949,982178,1075175
BC00518=87949,982178,1075175
BC00519=87949,982178,1075175
